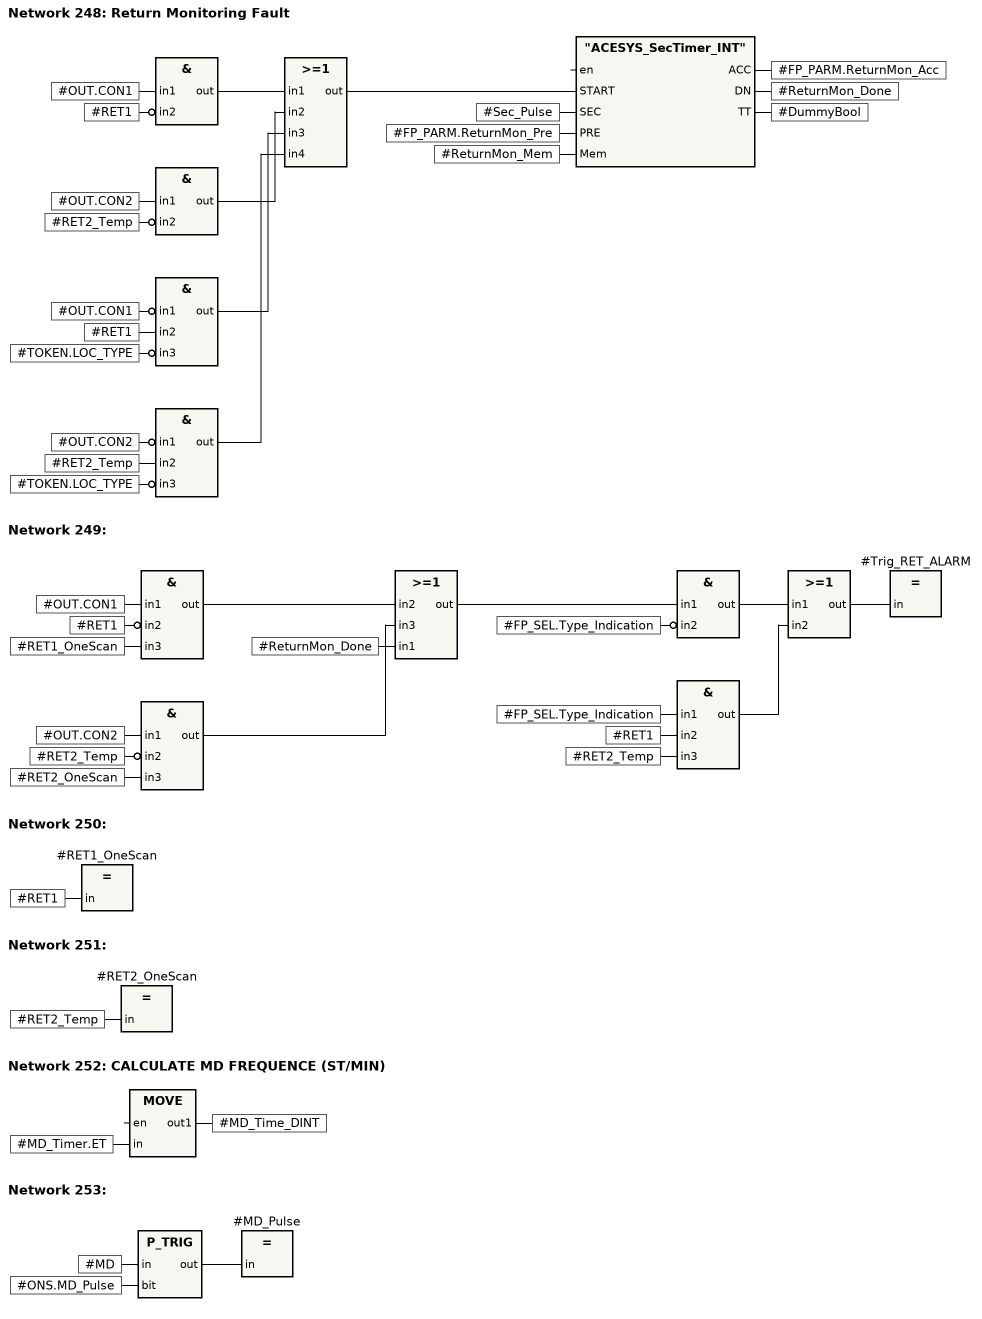
   "ACESYS_SecTimer_INT"(START := (#OUT.CON1 AND NOT #RET1) OR (#OUT.CON2 AND NOT #RET2_Temp) OR (NOT #OUT.CON1 AND #RET1 AND NOT #TOKEN.LOC_TYPE) OR (NOT #OUT.CON2 AND #RET2_Temp AND NOT #TOKEN.LOC_TYPE),
                         SEC := #Sec_Pulse,
                         PRE := #FP_PARM.ReturnMon_Pre,
                         Mem := #ReturnMon_Mem,
                         ACC => #FP_PARM.ReturnMon_Acc,
                         DN => #ReturnMon_Done,
                         TT => #DummyBool);
END_REGION

REGION Network 249
   #Trig_RET_ALARM := (((#OUT.CON1 AND NOT #RET1 AND #RET1_OneScan) OR (#OUT.CON2 AND NOT #RET2_Temp AND #RET2_OneScan) OR #ReturnMon_Done) AND NOT #FP_SEL.Type_Indication) OR (#FP_SEL.Type_Indication AND #RET1 AND #RET2_Temp);
END_REGION

REGION Network 250
   #RET1_OneScan := #RET1;
END_REGION

REGION Network 251
   #RET2_OneScan := #RET2_Temp;
END_REGION

REGION Network 252: CALCULATE MD FREQUENCE (ST/MIN)
   #MD_Time_DINT := #MD_Timer.ET;
END_REGION

REGION Network 253
   #_w1 := #MD AND NOT #ONS.MD_Pulse;   // rising edge
   #ONS.MD_Pulse := #MD;
   #MD_Pulse := #_w1;
END_REGION

REGION Network 254
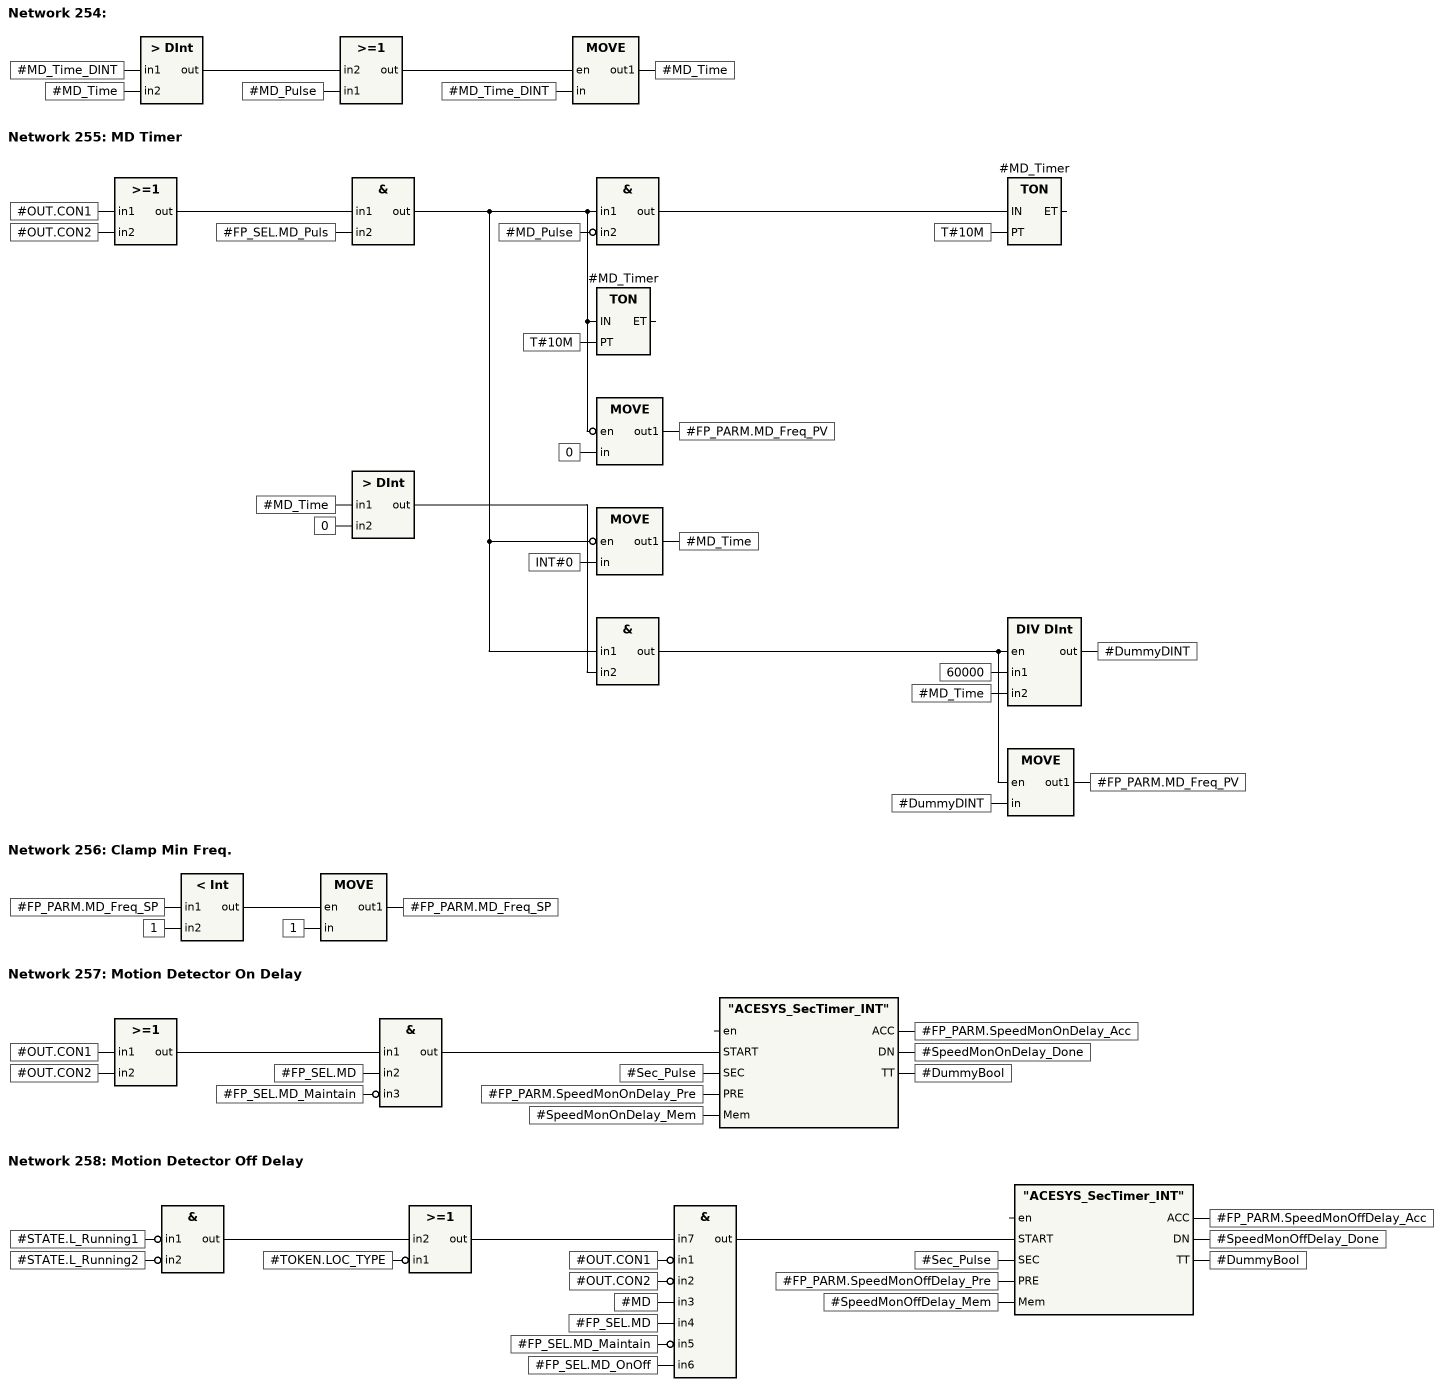
   IF (#MD_Time_DINT > #MD_Time) OR #MD_Pulse THEN #MD_Time := #MD_Time_DINT; END_IF;
END_REGION

REGION Network 255: MD Timer
   // The MD_Timer is inserted twice to ensure that the timer is enabled in the same 
   // scan after af MD pulse.
   #_w1 := (#OUT.CON1 OR #OUT.CON2) AND #FP_SEL.MD_Puls;
   #MD_Timer(IN := #_w1 AND NOT #MD_Pulse, PT := T#10M);   // TON
   #MD_Timer(IN := #_w1, PT := T#10M);   // TON
   IF NOT #_w1 THEN
       #FP_PARM.MD_Freq_PV := 0;
       #MD_Time := INT#0;
   END_IF;
   IF #_w1 AND (#MD_Time > 0) THEN
       #DummyDINT := 60000 / #MD_Time;
       #FP_PARM.MD_Freq_PV := #DummyDINT;
   END_IF;
END_REGION

REGION Network 256: Clamp Min Freq.
   IF #FP_PARM.MD_Freq_SP < 1 THEN #FP_PARM.MD_Freq_SP := 1; END_IF;
END_REGION

REGION Network 257: Motion Detector On Delay
   "ACESYS_SecTimer_INT"(START := (#OUT.CON1 OR #OUT.CON2) AND #FP_SEL.MD AND NOT #FP_SEL.MD_Maintain,
                         SEC := #Sec_Pulse,
                         PRE := #FP_PARM.SpeedMonOnDelay_Pre,
                         Mem := #SpeedMonOnDelay_Mem,
                         ACC => #FP_PARM.SpeedMonOnDelay_Acc,
                         DN => #SpeedMonOnDelay_Done,
                         TT => #DummyBool);
END_REGION

REGION Network 258: Motion Detector Off Delay
   // Build 003 - 1.July.2019 (EXTBOB): Added logic to inhibit motion fault when running in "electrical" local mode.
   "ACESYS_SecTimer_INT"(START := ((NOT #STATE.L_Running1 AND NOT #STATE.L_Running2) OR NOT #TOKEN.LOC_TYPE) AND NOT #OUT.CON1 AND NOT #OUT.CON2 AND #MD AND #FP_SEL.MD AND NOT #FP_SEL.MD_Maintain AND #FP_SEL.MD_OnOff,
                         SEC := #Sec_Pulse,
                         PRE := #FP_PARM.SpeedMonOffDelay_Pre,
                         Mem := #SpeedMonOffDelay_Mem,
                         ACC => #FP_PARM.SpeedMonOffDelay_Acc,
                         DN => #SpeedMonOffDelay_Done,
                         TT => #DummyBool);
END_REGION

REGION Network 259: Motion Detector Trig Delay
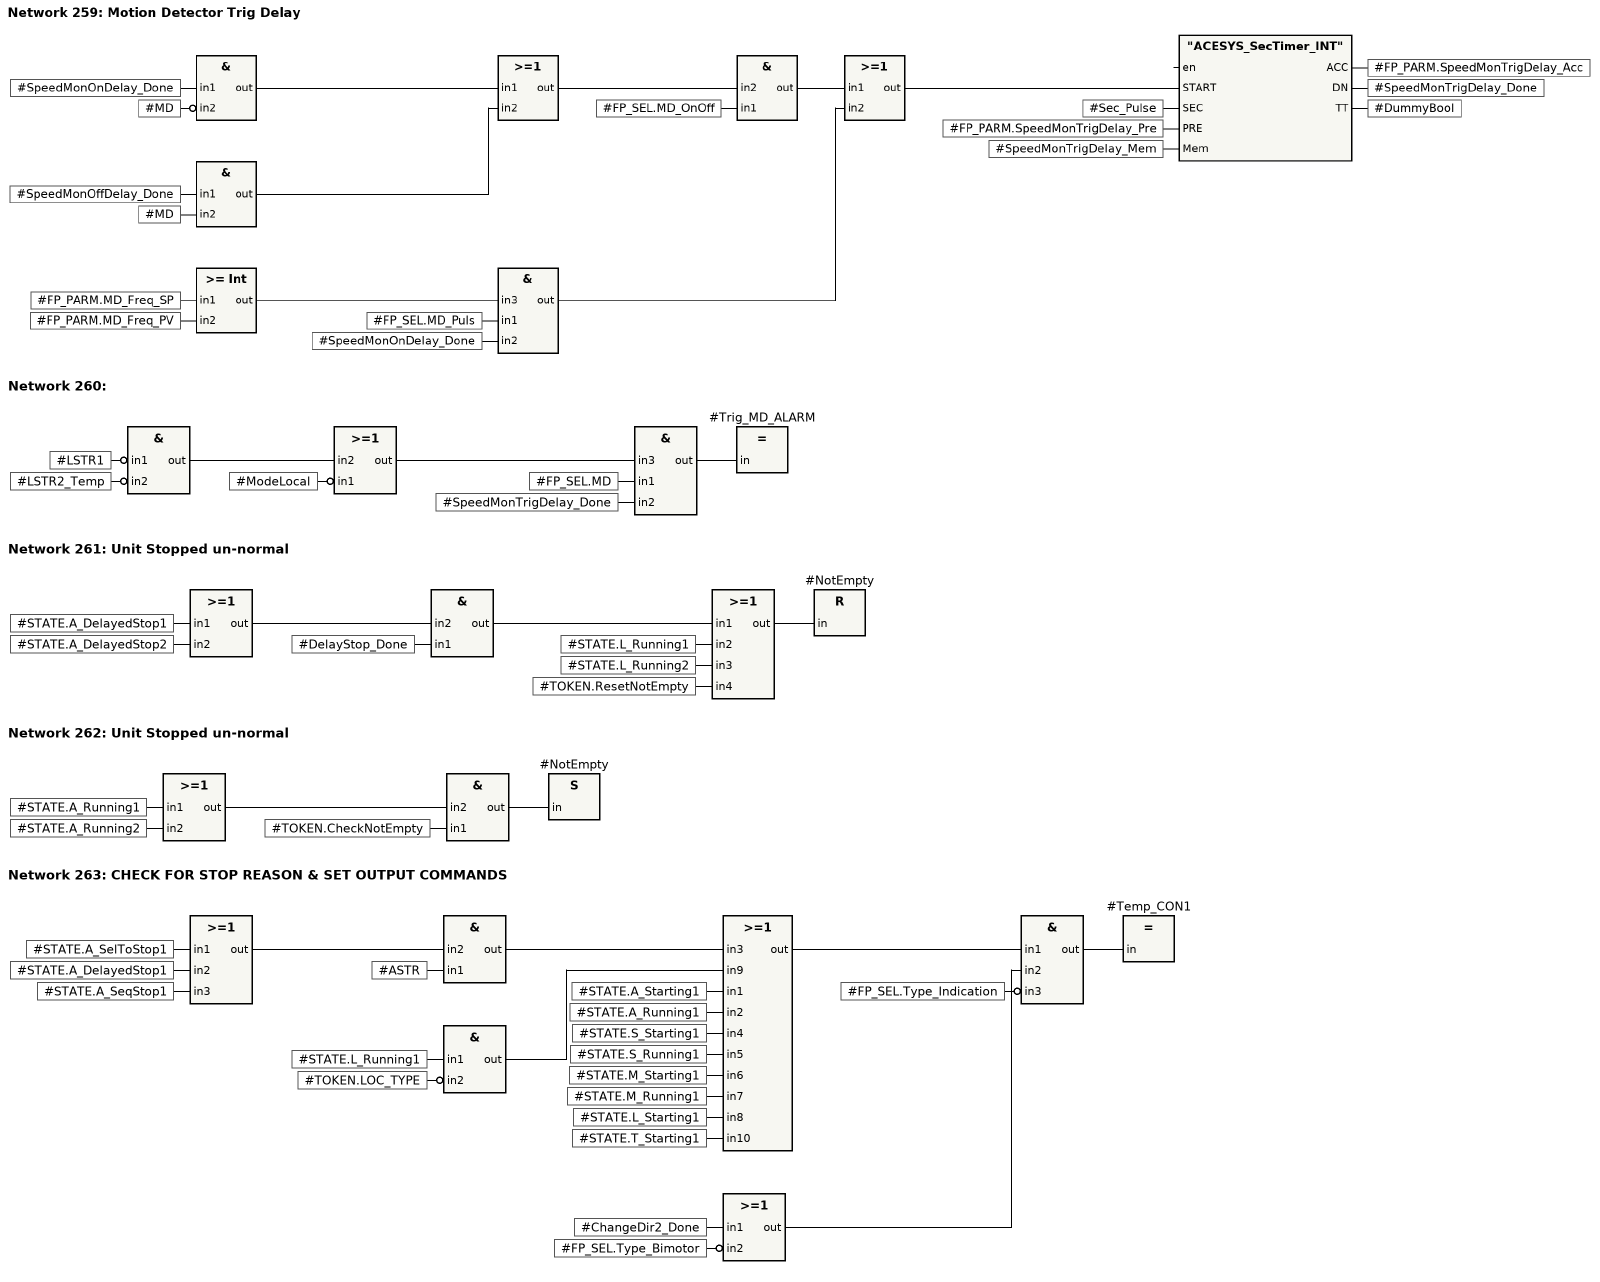
   "ACESYS_SecTimer_INT"(START := (((#SpeedMonOnDelay_Done AND NOT #MD) OR (#SpeedMonOffDelay_Done AND #MD)) AND #FP_SEL.MD_OnOff) OR ((#FP_PARM.MD_Freq_SP >= #FP_PARM.MD_Freq_PV) AND #FP_SEL.MD_Puls AND #SpeedMonOnDelay_Done),
                         SEC := #Sec_Pulse,
                         PRE := #FP_PARM.SpeedMonTrigDelay_Pre,
                         Mem := #SpeedMonTrigDelay_Mem,
                         ACC => #FP_PARM.SpeedMonTrigDelay_Acc,
                         DN => #SpeedMonTrigDelay_Done,
                         TT => #DummyBool);
END_REGION

REGION Network 260
   #Trig_MD_ALARM := ((NOT #LSTR1 AND NOT #LSTR2_Temp) OR NOT #ModeLocal) AND #FP_SEL.MD AND #SpeedMonTrigDelay_Done;
END_REGION

REGION Network 261: Unit Stopped un-normal
   // CHECK FOR MATERIANL IN LINE (NOT EMPTY)
   IF ((#STATE.A_DelayedStop1 OR #STATE.A_DelayedStop2) AND #DelayStop_Done) OR #STATE.L_Running1 OR #STATE.L_Running2 OR #TOKEN.ResetNotEmpty THEN
       #NotEmpty := FALSE;
   END_IF;
END_REGION

REGION Network 262: Unit Stopped un-normal
   // OK & INTL flags are replaced with A_Running1/2 flags
   IF (#STATE.A_Running1 OR #STATE.A_Running2) AND #TOKEN.CheckNotEmpty THEN #NotEmpty := TRUE; END_IF;
END_REGION

REGION Network 263: CHECK FOR STOP REASON & SET OUTPUT COMMANDS
   #Temp_CON1 := (((#STATE.A_SelToStop1 OR #STATE.A_DelayedStop1 OR #STATE.A_SeqStop1) AND #ASTR) OR (#STATE.L_Running1 AND NOT #TOKEN.LOC_TYPE) OR #STATE.A_Starting1 OR #STATE.A_Running1 OR #STATE.S_Starting1 OR #STATE.S_Running1 OR #STATE.M_Starting1 OR #STATE.M_Running1 OR #STATE.L_Starting1 OR #STATE.T_Starting1) AND (#ChangeDir2_Done OR NOT #FP_SEL.Type_Bimotor) AND NOT #FP_SEL.Type_Indication;
END_REGION

REGION Network 264
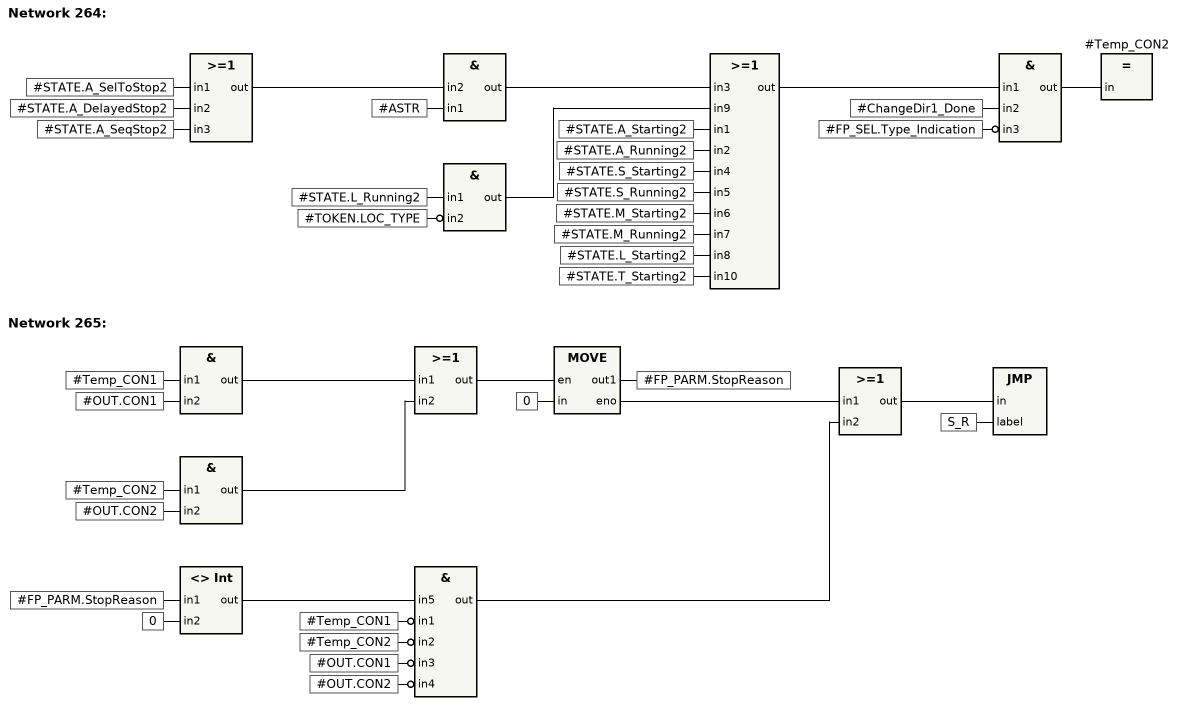
   #Temp_CON2 := (((#STATE.A_SelToStop2 OR #STATE.A_DelayedStop2 OR #STATE.A_SeqStop2) AND #ASTR) OR (#STATE.L_Running2 AND NOT #TOKEN.LOC_TYPE) OR #STATE.A_Starting2 OR #STATE.A_Running2 OR #STATE.S_Starting2 OR #STATE.S_Running2 OR #STATE.M_Starting2 OR #STATE.M_Running2 OR #STATE.L_Starting2 OR #STATE.T_Starting2) AND #ChangeDir1_Done AND NOT #FP_SEL.Type_Indication;
END_REGION

REGION Network 265
   // ENO of a box is taken as its EN; it also drops when the box reports an error
   #_w1 := (#Temp_CON1 AND #OUT.CON1) OR (#Temp_CON2 AND #OUT.CON2);
   IF #_w1 THEN #FP_PARM.StopReason := 0; END_IF;
   IF #_w1 OR ((#FP_PARM.StopReason <> 0) AND NOT #Temp_CON1 AND NOT #Temp_CON2 AND NOT #OUT.CON1 AND NOT #OUT.CON2) THEN
       GOTO S_R;
   END_IF;
END_REGION

REGION Network 266: Stop Reason
   // 0=In Operation
   // 1=Normal Stop
   // 2=Quick Stop
   // 3=Faceplate Stop
   // 4=Local Stop
   // 5=Change To Auto Mode
   // 6=Quick Stop From Unit Faceplate
   // 9=Sequence Interlock
   // 10=Interlock
   // 11=Unit Alarm
   // 12=Emergency Stop
   // 99=Unknown Reason
   // 
   // Build 003 - 8.July.2019 (EXTBOB): Stop Reason when ASTR goes low implemented
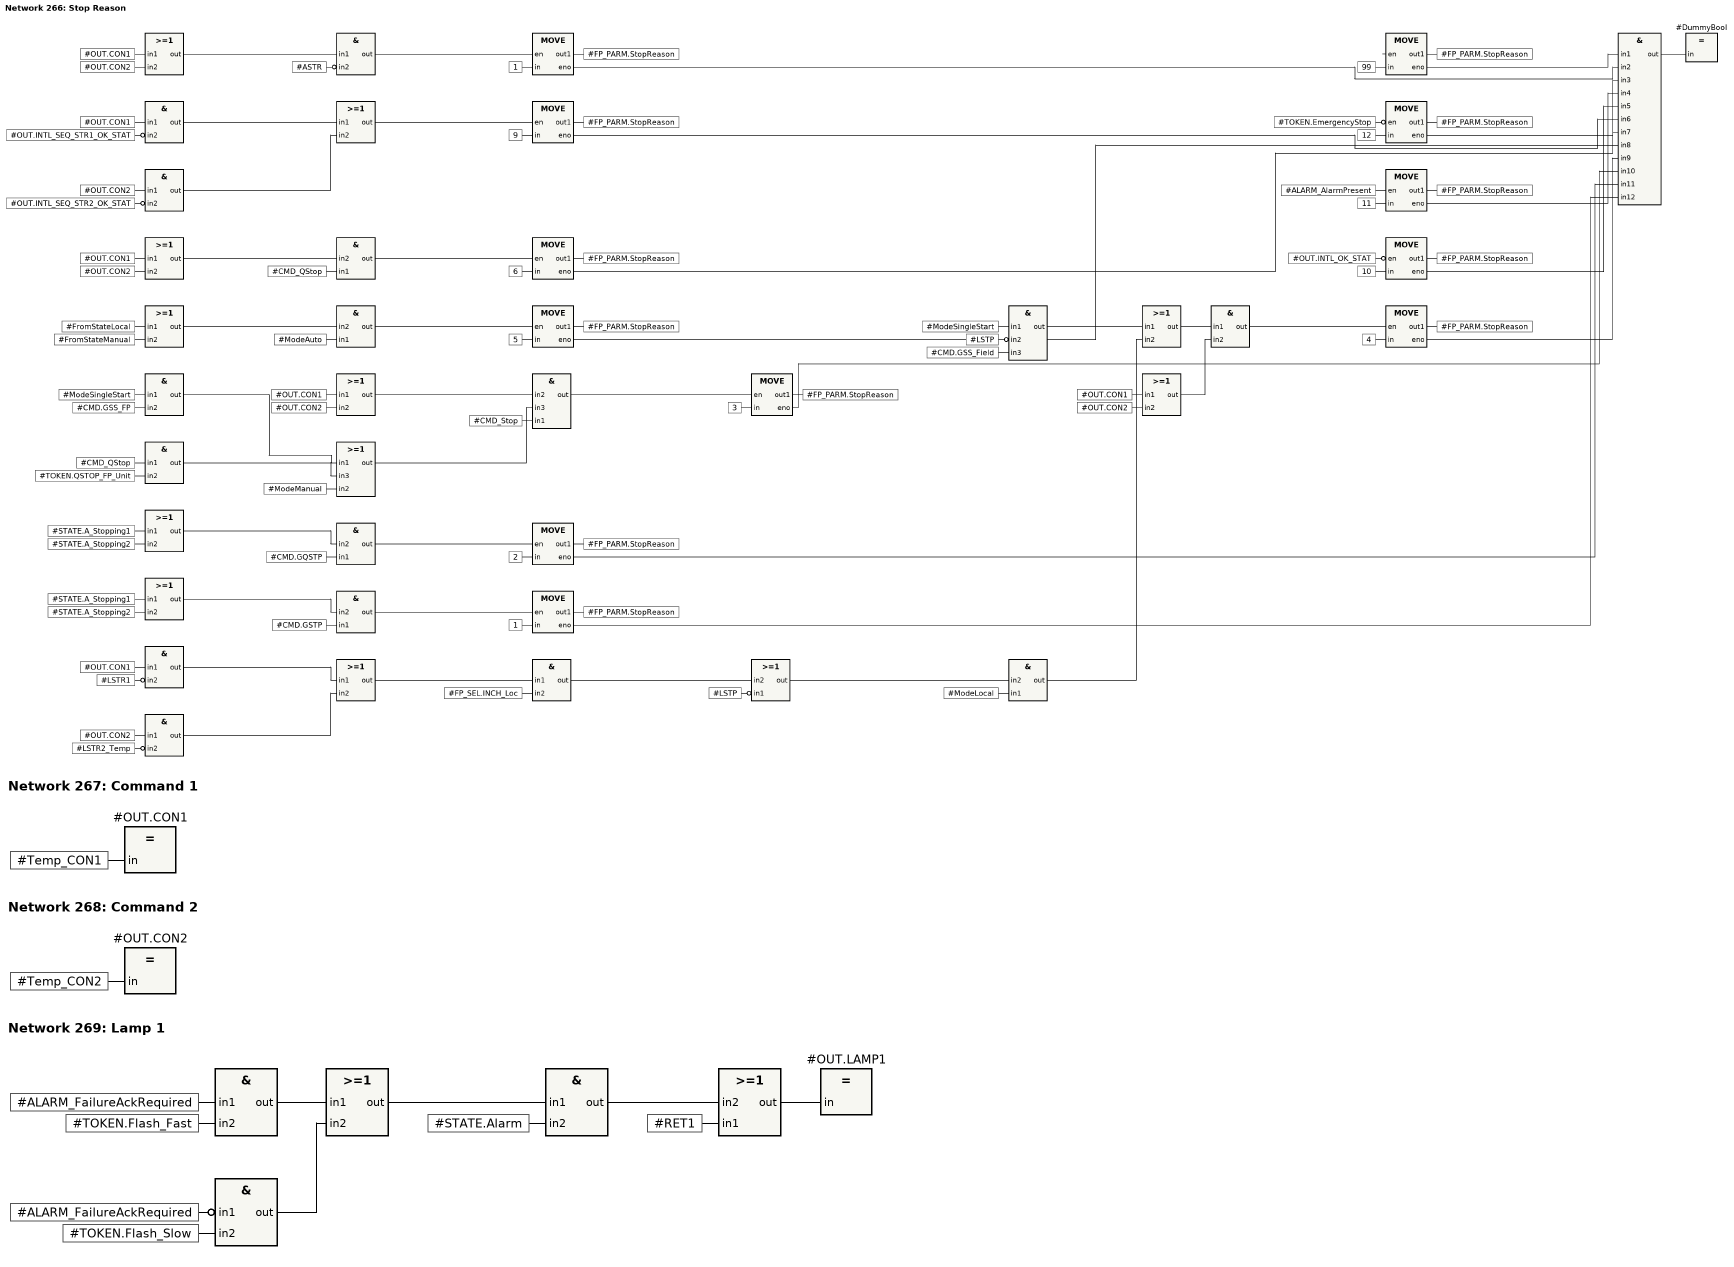
   // ENO of a box is taken as its EN; it also drops when the box reports an error
   #FP_PARM.StopReason := 99;
   #_w1 := (#OUT.CON1 OR #OUT.CON2) AND NOT #ASTR;
   IF #_w1 THEN #FP_PARM.StopReason := 1; END_IF;
   IF NOT #TOKEN.EmergencyStop THEN #FP_PARM.StopReason := 12; END_IF;
   IF #ALARM_AlarmPresent THEN #FP_PARM.StopReason := 11; END_IF;
   IF NOT #OUT.INTL_OK_STAT THEN #FP_PARM.StopReason := 10; END_IF;
   #_w2 := (#OUT.CON1 AND NOT #OUT.INTL_SEQ_STR1_OK_STAT) OR (#OUT.CON2 AND NOT #OUT.INTL_SEQ_STR2_OK_STAT);
   IF #_w2 THEN #FP_PARM.StopReason := 9; END_IF;
   #_w3 := (#OUT.CON1 OR #OUT.CON2) AND #CMD_QStop;
   IF #_w3 THEN #FP_PARM.StopReason := 6; END_IF;
   #_w4 := (#FromStateLocal OR #FromStateManual) AND #ModeAuto;
   IF #_w4 THEN #FP_PARM.StopReason := 5; END_IF;
   #_w5 := ((#ModeSingleStart AND NOT #LSTP AND #CMD.GSS_Field) OR (((((#OUT.CON1 AND NOT #LSTR1) OR (#OUT.CON2 AND NOT #LSTR2_Temp)) AND #FP_SEL.INCH_Loc) OR NOT #LSTP) AND #ModeLocal)) AND (#OUT.CON1 OR #OUT.CON2);
   IF #_w5 THEN #FP_PARM.StopReason := 4; END_IF;
   #_w6 := (#OUT.CON1 OR #OUT.CON2) AND ((#ModeSingleStart AND #CMD.GSS_FP) OR (#CMD_QStop AND #TOKEN.QSTOP_FP_Unit) OR #ModeManual) AND #CMD_Stop;
   IF #_w6 THEN #FP_PARM.StopReason := 3; END_IF;
   #_w7 := (#STATE.A_Stopping1 OR #STATE.A_Stopping2) AND #CMD.GQSTP;
   IF #_w7 THEN #FP_PARM.StopReason := 2; END_IF;
   #_w8 := (#STATE.A_Stopping1 OR #STATE.A_Stopping2) AND #CMD.GSTP;
   IF #_w8 THEN #FP_PARM.StopReason := 1; END_IF;
   #DummyBool := #_w1 AND NOT #TOKEN.EmergencyStop AND #ALARM_AlarmPresent AND NOT #OUT.INTL_OK_STAT AND #_w2 AND #_w3 AND #_w4 AND #_w5 AND #_w6 AND #_w7 AND #_w8;
END_REGION

REGION Network 267: Command 1
   S_R:
   #OUT.CON1 := #Temp_CON1;
END_REGION

REGION Network 268: Command 2
   #OUT.CON2 := #Temp_CON2;
END_REGION

REGION Network 269: Lamp 1
   // OUTPUT
   #OUT.LAMP1 := (((#ALARM_FailureAckRequired AND #TOKEN.Flash_Fast) OR (NOT #ALARM_FailureAckRequired AND #TOKEN.Flash_Slow)) AND #STATE.Alarm) OR #RET1;
END_REGION

REGION Network 270: Lamp 2
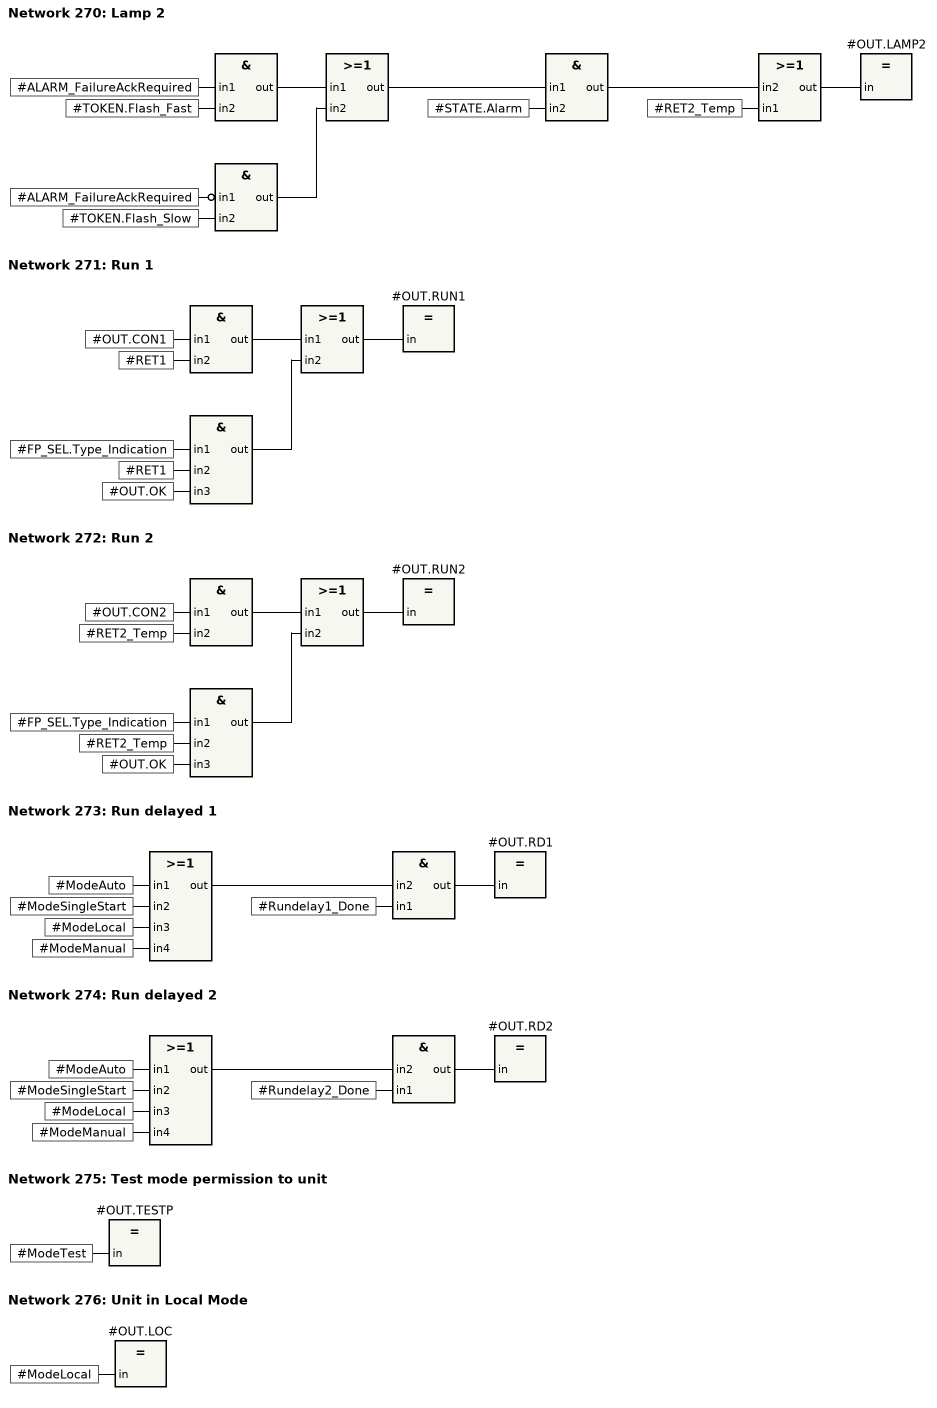
   #OUT.LAMP2 := (((#ALARM_FailureAckRequired AND #TOKEN.Flash_Fast) OR (NOT #ALARM_FailureAckRequired AND #TOKEN.Flash_Slow)) AND #STATE.Alarm) OR #RET2_Temp;
END_REGION

REGION Network 271: Run 1
   #OUT.RUN1 := (#OUT.CON1 AND #RET1) OR (#FP_SEL.Type_Indication AND #RET1 AND #OUT.OK);
END_REGION

REGION Network 272: Run 2
   #OUT.RUN2 := (#OUT.CON2 AND #RET2_Temp) OR (#FP_SEL.Type_Indication AND #RET2_Temp AND #OUT.OK);
END_REGION

REGION Network 273: Run delayed 1
   #OUT.RD1 := (#ModeAuto OR #ModeSingleStart OR #ModeLocal OR #ModeManual) AND #Rundelay1_Done;
END_REGION

REGION Network 274: Run delayed 2
   #OUT.RD2 := (#ModeAuto OR #ModeSingleStart OR #ModeLocal OR #ModeManual) AND #Rundelay2_Done;
END_REGION

REGION Network 275: Test mode permission to unit
   #OUT.TESTP := #ModeTest;
END_REGION

REGION Network 276: Unit in Local Mode
   #OUT.LOC := #ModeLocal;
END_REGION

REGION Network 277: Unit in Manual Mode
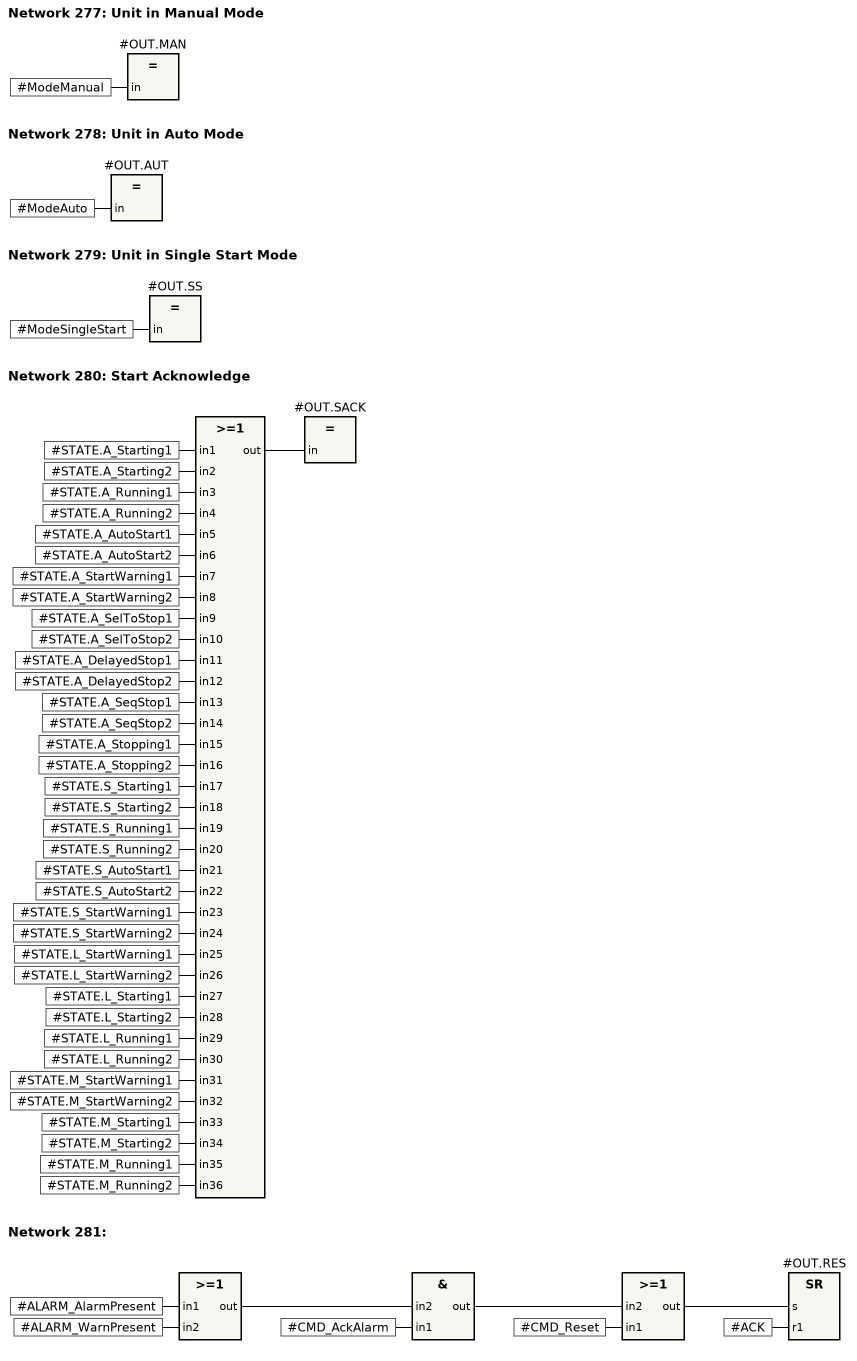
   #OUT.MAN := #ModeManual;
END_REGION

REGION Network 278: Unit in Auto Mode
   #OUT.AUT := #ModeAuto;
END_REGION

REGION Network 279: Unit in Single Start Mode
   #OUT.SS := #ModeSingleStart;
END_REGION

REGION Network 280: Start Acknowledge
   #OUT.SACK := #STATE.A_Starting1 OR #STATE.A_Starting2 OR #STATE.A_Running1 OR #STATE.A_Running2 OR #STATE.A_AutoStart1 OR #STATE.A_AutoStart2 OR #STATE.A_StartWarning1 OR #STATE.A_StartWarning2 OR #STATE.A_SelToStop1 OR #STATE.A_SelToStop2 OR #STATE.A_DelayedStop1 OR #STATE.A_DelayedStop2 OR #STATE.A_SeqStop1 OR #STATE.A_SeqStop2 OR #STATE.A_Stopping1 OR #STATE.A_Stopping2 OR #STATE.S_Starting1 OR #STATE.S_Starting2 OR #STATE.S_Running1 OR #STATE.S_Running2 OR #STATE.S_AutoStart1 OR #STATE.S_AutoStart2 OR #STATE.S_StartWarning1 OR #STATE.S_StartWarning2 OR #STATE.L_StartWarning1 OR #STATE.L_StartWarning2 OR #STATE.L_Starting1 OR #STATE.L_Starting2 OR #STATE.L_Running1 OR #STATE.L_Running2 OR #STATE.M_StartWarning1 OR #STATE.M_StartWarning2 OR #STATE.M_Starting1 OR #STATE.M_Starting2 OR #STATE.M_Running1 OR #STATE.M_Running2;
END_REGION

REGION Network 281
   IF ((#ALARM_AlarmPresent OR #ALARM_WarnPresent) AND #CMD_AckAlarm) OR #CMD_Reset THEN
       #OUT.RES := TRUE;   // SR flip-flop
   END_IF;
   IF #ACK THEN #OUT.RES := FALSE; END_IF;
END_REGION

REGION Network 282: Unit Status OK (no alarms)
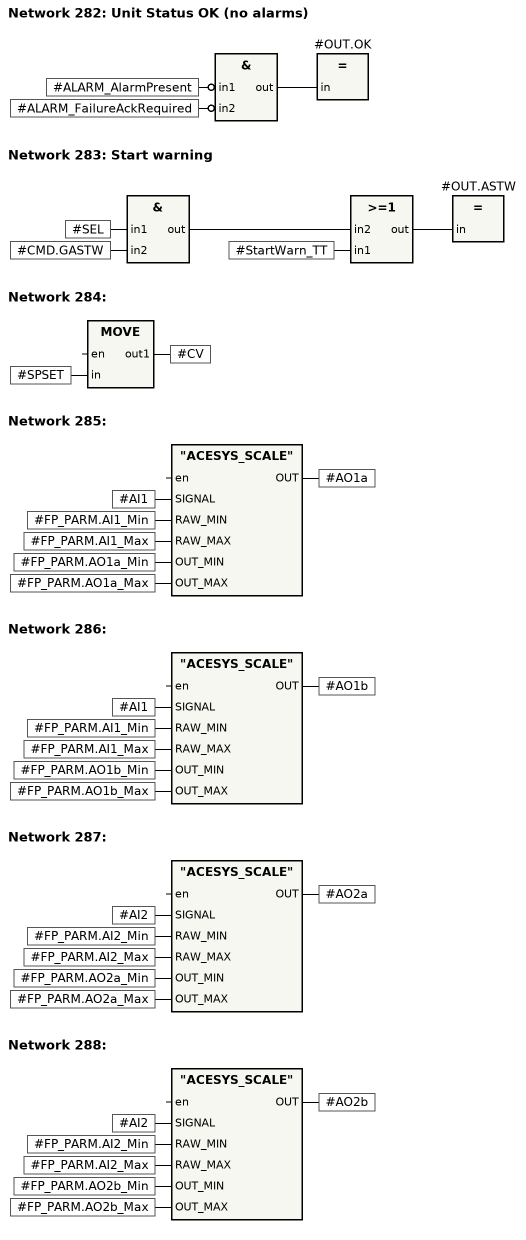
   #OUT.OK := NOT #ALARM_AlarmPresent AND NOT #ALARM_FailureAckRequired;
END_REGION

REGION Network 283: Start warning
   #OUT.ASTW := (#SEL AND #CMD.GASTW) OR #StartWarn_TT;
END_REGION

REGION Network 284
   #CV := #SPSET;
END_REGION

REGION Network 285
   "ACESYS_SCALE"(SIGNAL := #AI1,
                  RAW_MIN := #FP_PARM.AI1_Min,
                  RAW_MAX := #FP_PARM.AI1_Max,
                  OUT_MIN := #FP_PARM.AO1a_Min,
                  OUT_MAX := #FP_PARM.AO1a_Max,
                  OUT => #AO1a);
END_REGION

REGION Network 286
   "ACESYS_SCALE"(SIGNAL := #AI1,
                  RAW_MIN := #FP_PARM.AI1_Min,
                  RAW_MAX := #FP_PARM.AI1_Max,
                  OUT_MIN := #FP_PARM.AO1b_Min,
                  OUT_MAX := #FP_PARM.AO1b_Max,
                  OUT => #AO1b);
END_REGION

REGION Network 287
   "ACESYS_SCALE"(SIGNAL := #AI2,
                  RAW_MIN := #FP_PARM.AI2_Min,
                  RAW_MAX := #FP_PARM.AI2_Max,
                  OUT_MIN := #FP_PARM.AO2a_Min,
                  OUT_MAX := #FP_PARM.AO2a_Max,
                  OUT => #AO2a);
END_REGION

REGION Network 288
   "ACESYS_SCALE"(SIGNAL := #AI2,
                  RAW_MIN := #FP_PARM.AI2_Min,
                  RAW_MAX := #FP_PARM.AI2_Max,
                  OUT_MIN := #FP_PARM.AO2b_Min,
                  OUT_MAX := #FP_PARM.AO2b_Max,
                  OUT => #AO2b);
END_REGION

REGION Network 289
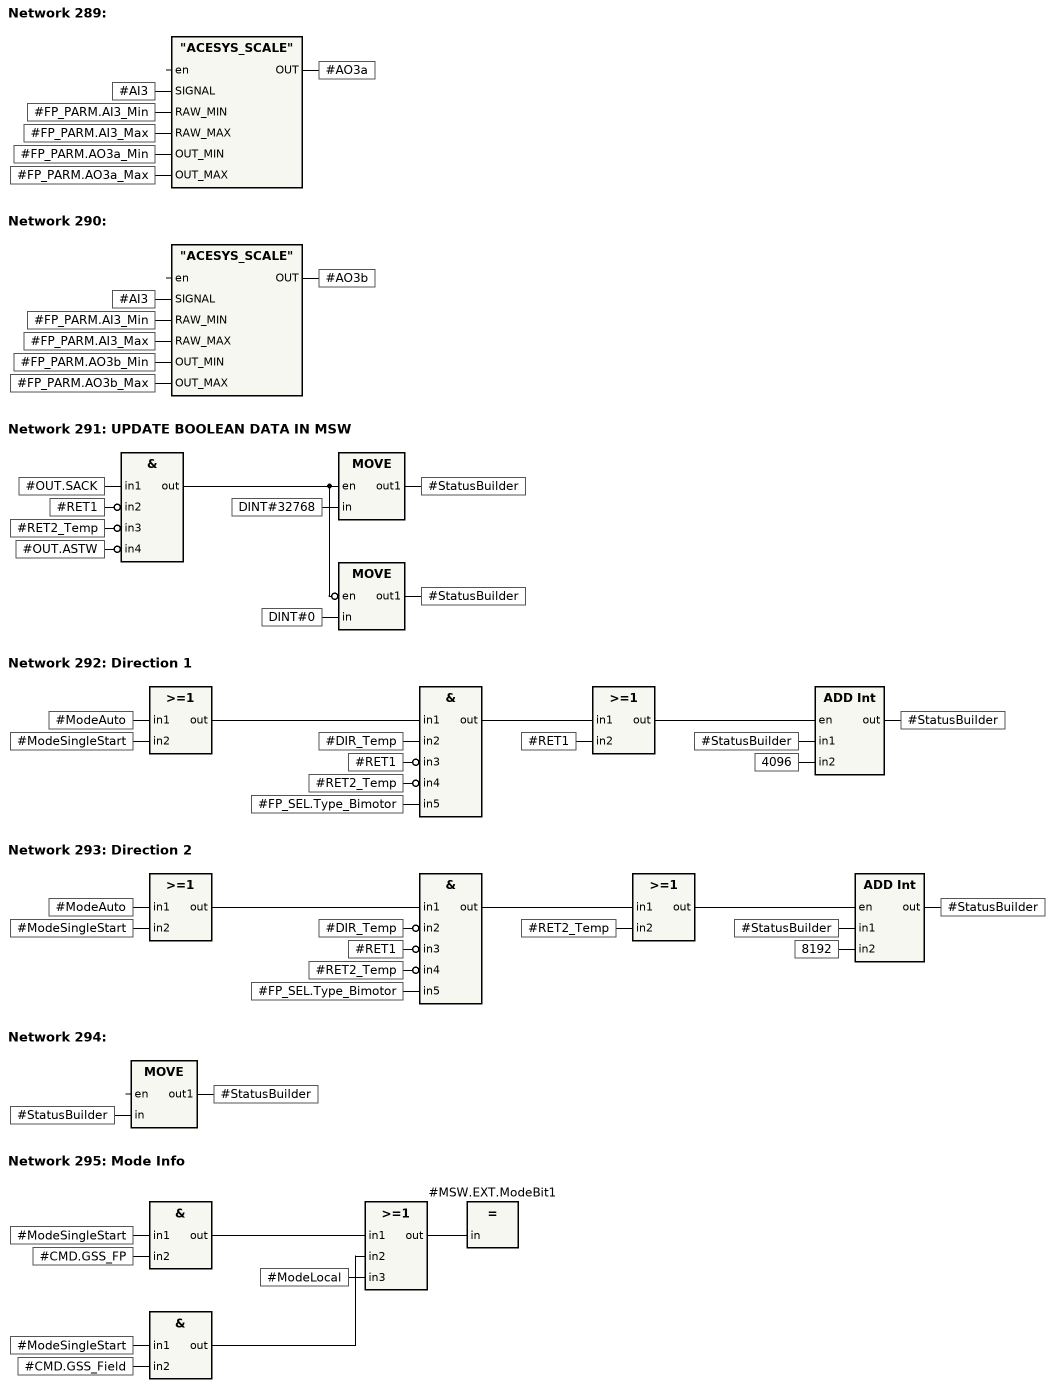
   "ACESYS_SCALE"(SIGNAL := #AI3,
                  RAW_MIN := #FP_PARM.AI3_Min,
                  RAW_MAX := #FP_PARM.AI3_Max,
                  OUT_MIN := #FP_PARM.AO3a_Min,
                  OUT_MAX := #FP_PARM.AO3a_Max,
                  OUT => #AO3a);
END_REGION

REGION Network 290
   "ACESYS_SCALE"(SIGNAL := #AI3,
                  RAW_MIN := #FP_PARM.AI3_Min,
                  RAW_MAX := #FP_PARM.AI3_Max,
                  OUT_MIN := #FP_PARM.AO3b_Min,
                  OUT_MAX := #FP_PARM.AO3b_Max,
                  OUT => #AO3b);
END_REGION

REGION Network 291: UPDATE BOOLEAN DATA IN MSW
   #_w1 := #OUT.SACK AND NOT #RET1 AND NOT #RET2_Temp AND NOT #OUT.ASTW;
   IF #_w1 THEN #StatusBuilder := DINT#32768; END_IF;
   IF NOT #_w1 THEN #StatusBuilder := DINT#0; END_IF;
END_REGION

REGION Network 292: Direction 1
   // Build 002 - 27 March 2019 - FP_Sel.Type_Bimotor Added
   IF ((#ModeAuto OR #ModeSingleStart) AND #DIR_Temp AND NOT #RET1 AND NOT #RET2_Temp AND #FP_SEL.Type_Bimotor) OR #RET1 THEN
       #StatusBuilder := #StatusBuilder + 4096;
   END_IF;
END_REGION

REGION Network 293: Direction 2
   // Build 002 - 27 March 2019 - FP_Sel.Type_Bimotor Added
   IF ((#ModeAuto OR #ModeSingleStart) AND NOT #DIR_Temp AND NOT #RET1 AND NOT #RET2_Temp AND #FP_SEL.Type_Bimotor) OR #RET2_Temp THEN
       #StatusBuilder := #StatusBuilder + 8192;
   END_IF;
END_REGION

REGION Network 294
   #StatusBuilder := #StatusBuilder;
END_REGION

REGION Network 295: Mode Info
   #MSW.EXT.ModeBit1 := (#ModeSingleStart AND #CMD.GSS_FP) OR (#ModeSingleStart AND #CMD.GSS_Field) OR #ModeLocal;
END_REGION

REGION Network 296: Mode Info
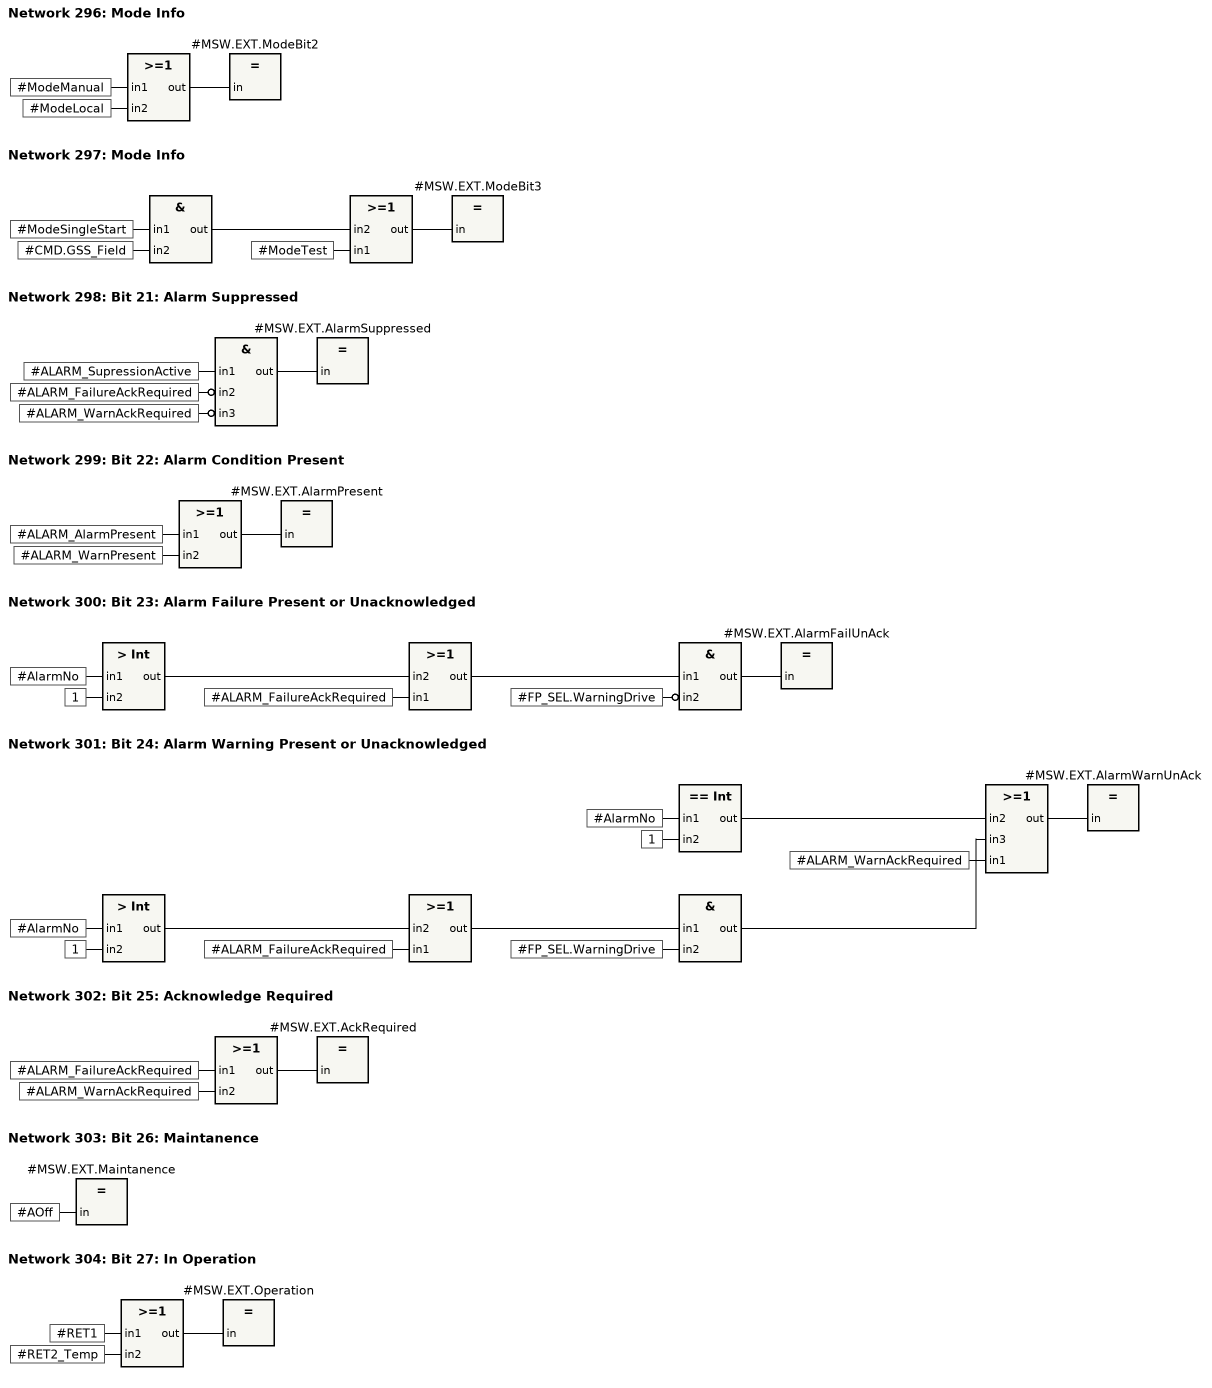
   #MSW.EXT.ModeBit2 := #ModeManual OR #ModeLocal;
END_REGION

REGION Network 297: Mode Info
   #MSW.EXT.ModeBit3 := (#ModeSingleStart AND #CMD.GSS_Field) OR #ModeTest;
END_REGION

REGION Network 298: Bit 21: Alarm Suppressed
   #MSW.EXT.AlarmSuppressed := #ALARM_SupressionActive AND NOT #ALARM_FailureAckRequired AND NOT #ALARM_WarnAckRequired;
END_REGION

REGION Network 299: Bit 22: Alarm Condition Present
   #MSW.EXT.AlarmPresent := #ALARM_AlarmPresent OR #ALARM_WarnPresent;
END_REGION

REGION Network 300: Bit 23: Alarm Failure Present or Unacknowledged
   #MSW.EXT.AlarmFailUnAck := ((#AlarmNo > 1) OR #ALARM_FailureAckRequired) AND NOT #FP_SEL.WarningDrive;
END_REGION

REGION Network 301: Bit 24: Alarm Warning Present or Unacknowledged
   #MSW.EXT.AlarmWarnUnAck := (#AlarmNo = 1) OR (((#AlarmNo > 1) OR #ALARM_FailureAckRequired) AND #FP_SEL.WarningDrive) OR #ALARM_WarnAckRequired;
END_REGION

REGION Network 302: Bit 25: Acknowledge Required
   #MSW.EXT.AckRequired := #ALARM_FailureAckRequired OR #ALARM_WarnAckRequired;
END_REGION

REGION Network 303: Bit 26: Maintanence
   #MSW.EXT.Maintanence := #AOff;
END_REGION

REGION Network 304: Bit 27: In Operation
   #MSW.EXT.Operation := #RET1 OR #RET2_Temp;
END_REGION

REGION Network 305: Bit 28: Forced
   // Build 002 - 25 March 2019 : Out of Service flag would set the Forced flag to 
   // symbols
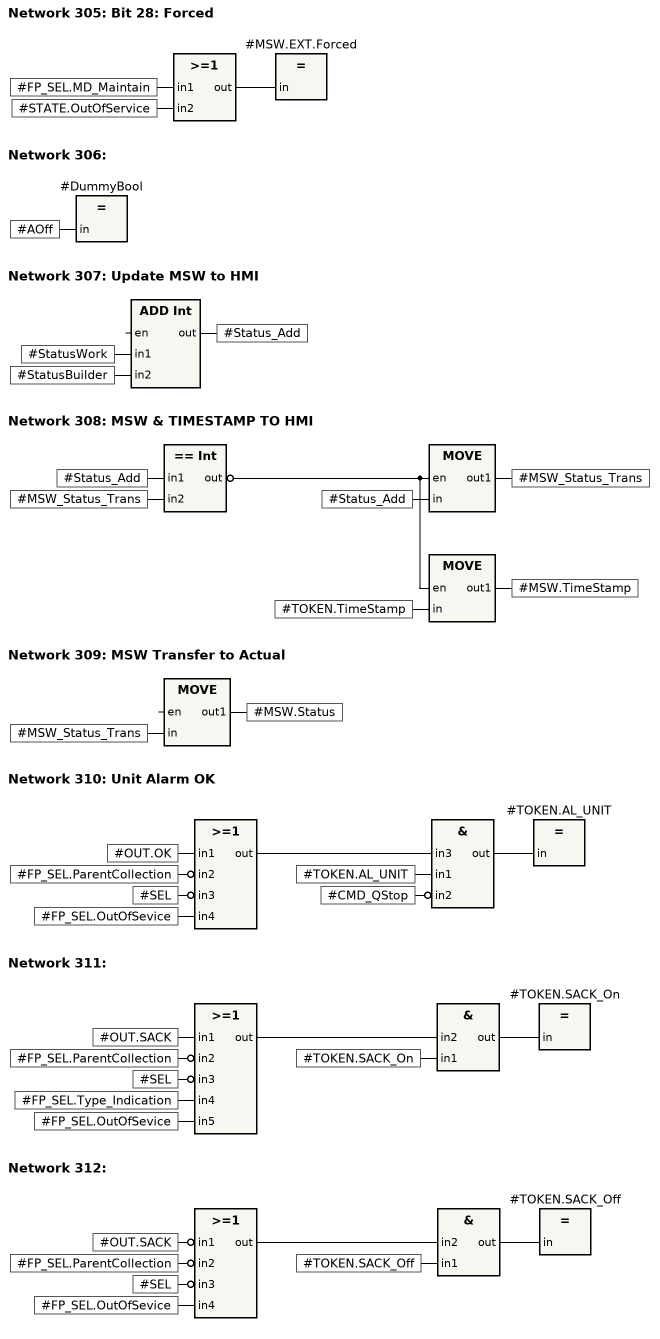
   #MSW.EXT.Forced := #FP_SEL.MD_Maintain OR #STATE.OutOfService;
END_REGION

REGION Network 306
   Done:
   #DummyBool := #AOff;
END_REGION

REGION Network 307: Update MSW to HMI
   #Status_Add := #StatusWork + #StatusBuilder;
END_REGION

REGION Network 308: MSW & TIMESTAMP TO HMI
   #_w1 := NOT (#Status_Add = #MSW_Status_Trans);
   IF #_w1 THEN
       #MSW_Status_Trans := #Status_Add;
       #MSW.TimeStamp := #TOKEN.TimeStamp;
   END_IF;
END_REGION

REGION Network 309: MSW Transfer to Actual
   #MSW.Status := #MSW_Status_Trans;
END_REGION

REGION Network 310: Unit Alarm OK
   #TOKEN.AL_UNIT := (#OUT.OK OR NOT #FP_SEL.ParentCollection OR NOT #SEL OR #FP_SEL.OutOfSevice) AND #TOKEN.AL_UNIT AND NOT #CMD_QStop;
END_REGION

REGION Network 311
   // Build 003 - 1.July.2019 (EXTBOB): Replaced "Select" with original explicit definition
   // Build 009 - 24.Jun.2020 (MIA-US): Remove CMD.GSEL
   #TOKEN.SACK_On := (#OUT.SACK OR NOT #FP_SEL.ParentCollection OR NOT #SEL OR #FP_SEL.Type_Indication OR #FP_SEL.OutOfSevice) AND #TOKEN.SACK_On;
END_REGION

REGION Network 312
   #TOKEN.SACK_Off := (NOT #OUT.SACK OR NOT #FP_SEL.ParentCollection OR NOT #SEL OR #FP_SEL.OutOfSevice) AND #TOKEN.SACK_Off;
END_REGION

REGION Network 313
   // Build 003 - 1.July.2019 (EXTBOB): Replaced "Select" with original explicit definition
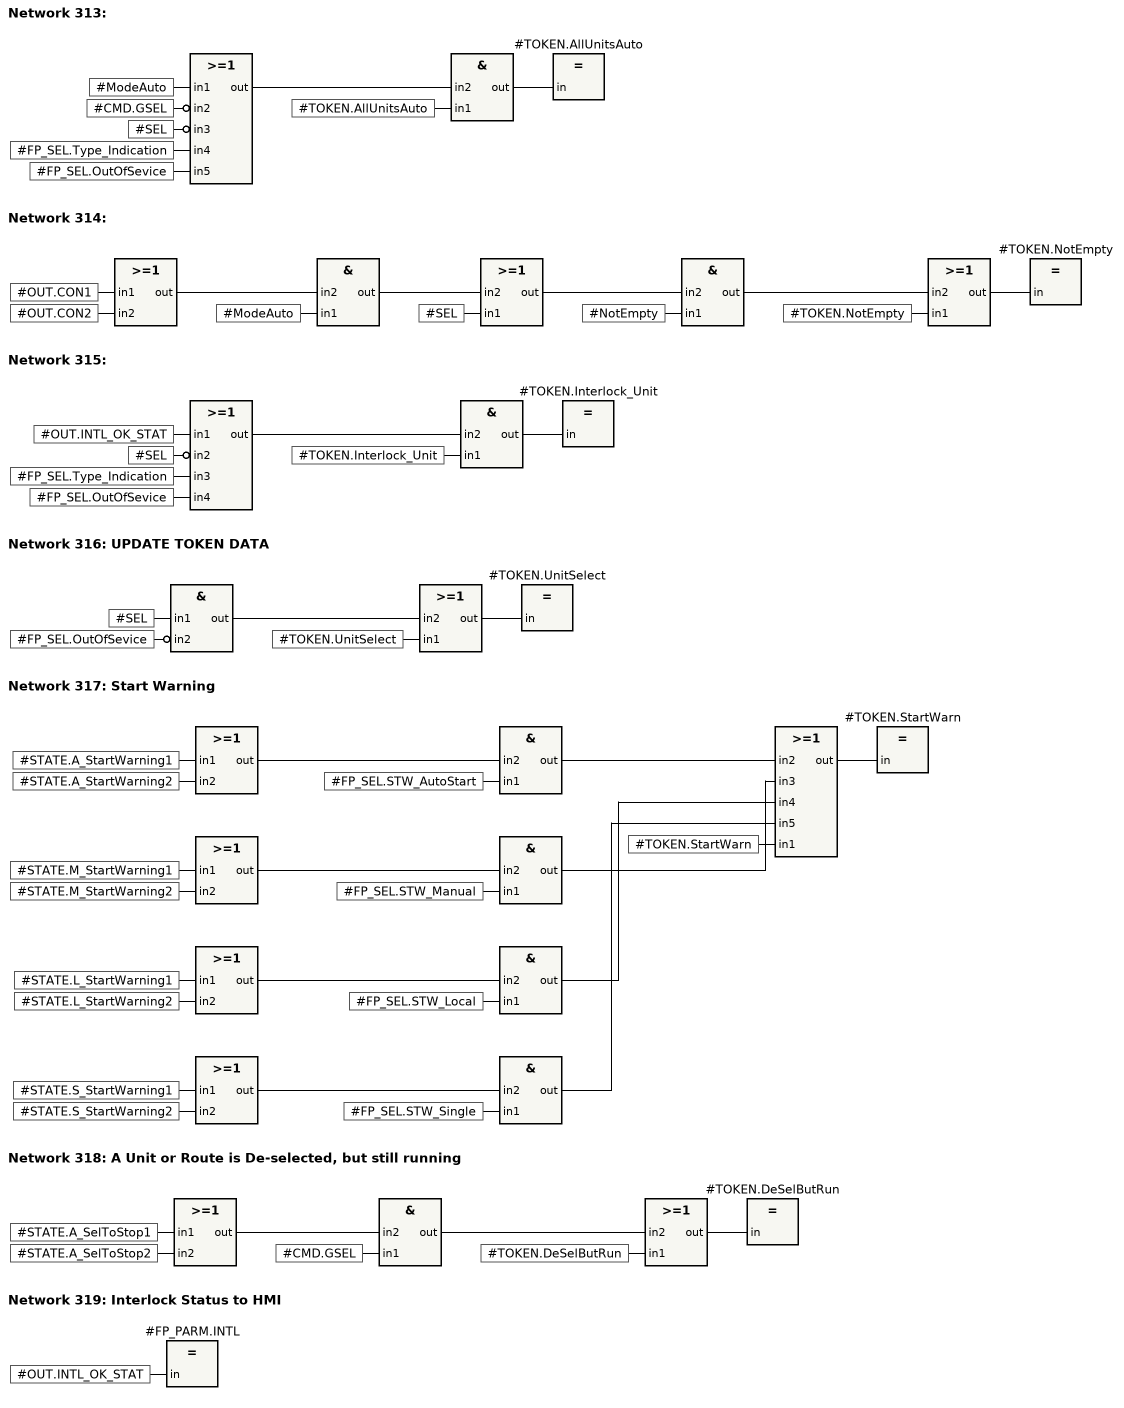
   #TOKEN.AllUnitsAuto := (#ModeAuto OR NOT #CMD.GSEL OR NOT #SEL OR #FP_SEL.Type_Indication OR #FP_SEL.OutOfSevice) AND #TOKEN.AllUnitsAuto;
END_REGION

REGION Network 314
   #TOKEN.NotEmpty := ((((#OUT.CON1 OR #OUT.CON2) AND #ModeAuto) OR #SEL) AND #NotEmpty) OR #TOKEN.NotEmpty;
END_REGION

REGION Network 315
   // Build 003 - 1.July.2019 (EXTBOB): Replaced "Select" with original explicit definition
   // Build 011 - 09.10.2020 (EXTBOB): Removed CMD.GSEL neg in OR logic to pass Intl status also in grp deselected cond in auto mode
   #TOKEN.Interlock_Unit := (#OUT.INTL_OK_STAT OR NOT #SEL OR #FP_SEL.Type_Indication OR #FP_SEL.OutOfSevice) AND #TOKEN.Interlock_Unit;
END_REGION

REGION Network 316: UPDATE TOKEN DATA
   #TOKEN.UnitSelect := (#SEL AND NOT #FP_SEL.OutOfSevice) OR #TOKEN.UnitSelect;
END_REGION

REGION Network 317: Start Warning
   #TOKEN.StartWarn := ((#STATE.A_StartWarning1 OR #STATE.A_StartWarning2) AND #FP_SEL.STW_AutoStart) OR ((#STATE.M_StartWarning1 OR #STATE.M_StartWarning2) AND #FP_SEL.STW_Manual) OR ((#STATE.L_StartWarning1 OR #STATE.L_StartWarning2) AND #FP_SEL.STW_Local) OR ((#STATE.S_StartWarning1 OR #STATE.S_StartWarning2) AND #FP_SEL.STW_Single) OR #TOKEN.StartWarn;
END_REGION

REGION Network 318: A Unit or Route is De-selected, but still running
   #TOKEN.DeSelButRun := ((#STATE.A_SelToStop1 OR #STATE.A_SelToStop2) AND #CMD.GSEL) OR #TOKEN.DeSelButRun;
END_REGION

REGION Network 319: Interlock Status to HMI
   #FP_PARM.INTL := #OUT.INTL_OK_STAT;
END_REGION

REGION Network 320: Interlock Status to HMI
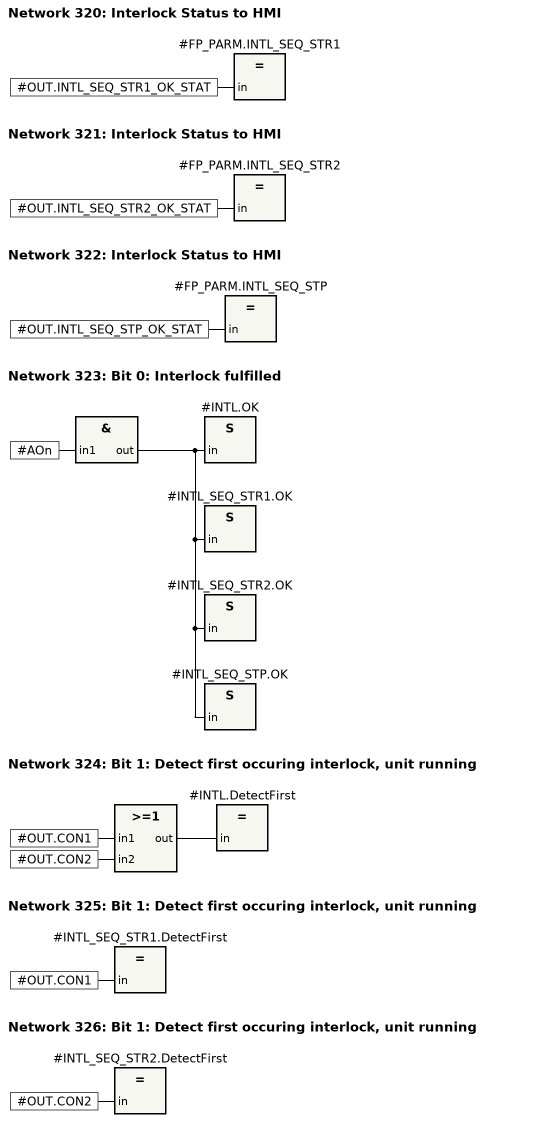
   #FP_PARM.INTL_SEQ_STR1 := #OUT.INTL_SEQ_STR1_OK_STAT;
END_REGION

REGION Network 321: Interlock Status to HMI
   #FP_PARM.INTL_SEQ_STR2 := #OUT.INTL_SEQ_STR2_OK_STAT;
END_REGION

REGION Network 322: Interlock Status to HMI
   #FP_PARM.INTL_SEQ_STP := #OUT.INTL_SEQ_STP_OK_STAT;
END_REGION

REGION Network 323: Bit 0: Interlock fulfilled
   // INTERLOCK LINK
   IF #AOn THEN
       #INTL.OK := TRUE;
       #INTL_SEQ_STR1.OK := TRUE;
       #INTL_SEQ_STR2.OK := TRUE;
       #INTL_SEQ_STP.OK := TRUE;
   END_IF;
END_REGION

REGION Network 324: Bit 1: Detect first occuring interlock, unit running
   #INTL.DetectFirst := #OUT.CON1 OR #OUT.CON2;
END_REGION

REGION Network 325: Bit 1: Detect first occuring interlock, unit running
   #INTL_SEQ_STR1.DetectFirst := #OUT.CON1;
END_REGION

REGION Network 326: Bit 1: Detect first occuring interlock, unit running
   #INTL_SEQ_STR2.DetectFirst := #OUT.CON2;
END_REGION

REGION Network 327: Bit 3: Clear first Interlock
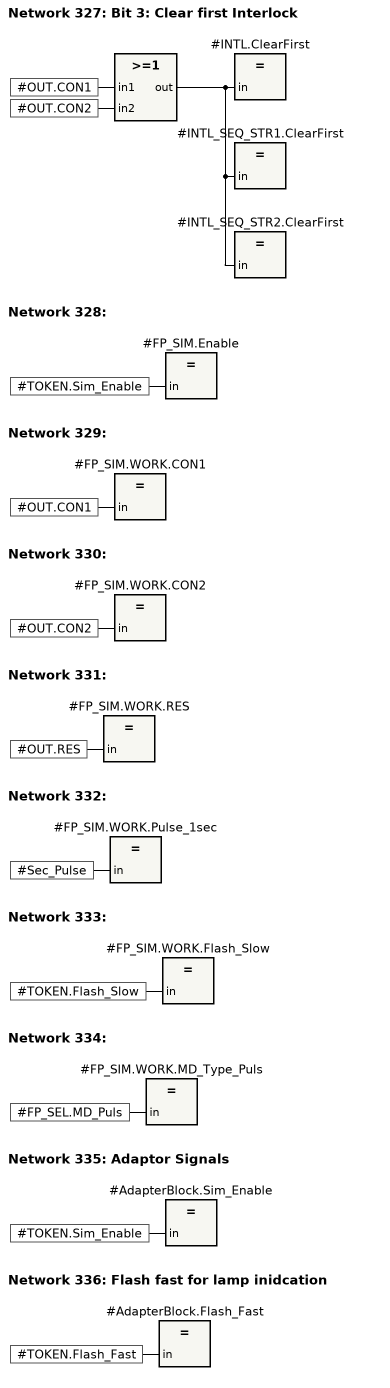
   #INTL.ClearFirst := #OUT.CON1 OR #OUT.CON2;
   #INTL_SEQ_STR1.ClearFirst := #INTL.ClearFirst;
   #INTL_SEQ_STR2.ClearFirst := #INTL.ClearFirst;
END_REGION

REGION Network 328
   #FP_SIM.Enable := #TOKEN.Sim_Enable;
END_REGION

REGION Network 329
   #FP_SIM.WORK.CON1 := #OUT.CON1;
END_REGION

REGION Network 330
   #FP_SIM.WORK.CON2 := #OUT.CON2;
END_REGION

REGION Network 331
   #FP_SIM.WORK.RES := #OUT.RES;
END_REGION

REGION Network 332
   #FP_SIM.WORK.Pulse_1sec := #Sec_Pulse;
END_REGION

REGION Network 333
   #FP_SIM.WORK.Flash_Slow := #TOKEN.Flash_Slow;
END_REGION

REGION Network 334
   #FP_SIM.WORK.MD_Type_Puls := #FP_SEL.MD_Puls;
END_REGION

REGION Network 335: Adaptor Signals
   #AdapterBlock.Sim_Enable := #TOKEN.Sim_Enable;
END_REGION

REGION Network 336: Flash fast for lamp inidcation
   #AdapterBlock.Flash_Fast := #TOKEN.Flash_Fast;
END_REGION

REGION Network 337: Flash slow for lamp inidcation
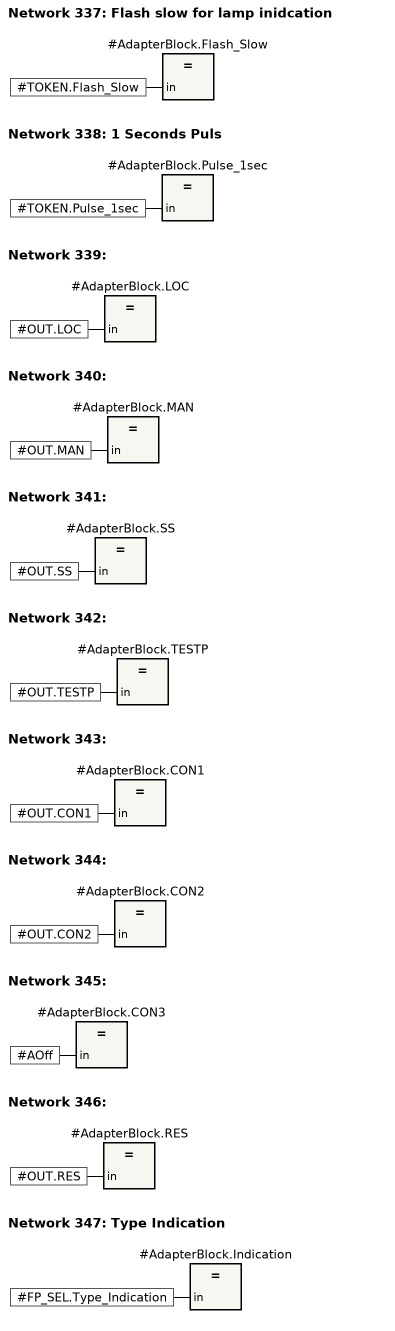
   #AdapterBlock.Flash_Slow := #TOKEN.Flash_Slow;
END_REGION

REGION Network 338: 1 Seconds Puls
   #AdapterBlock.Pulse_1sec := #TOKEN.Pulse_1sec;
END_REGION

REGION Network 339
   #AdapterBlock.LOC := #OUT.LOC;
END_REGION

REGION Network 340
   #AdapterBlock.MAN := #OUT.MAN;
END_REGION

REGION Network 341
   #AdapterBlock.SS := #OUT.SS;
END_REGION

REGION Network 342
   #AdapterBlock.TESTP := #OUT.TESTP;
END_REGION

REGION Network 343
   #AdapterBlock.CON1 := #OUT.CON1;
END_REGION

REGION Network 344
   #AdapterBlock.CON2 := #OUT.CON2;
END_REGION

REGION Network 345
   #AdapterBlock.CON3 := #AOff;
END_REGION

REGION Network 346
   #AdapterBlock.RES := #OUT.RES;
END_REGION

REGION Network 347: Type Indication
   #AdapterBlock.Indication := #FP_SEL.Type_Indication;
END_REGION

REGION Network 348: Write STAT to OUT
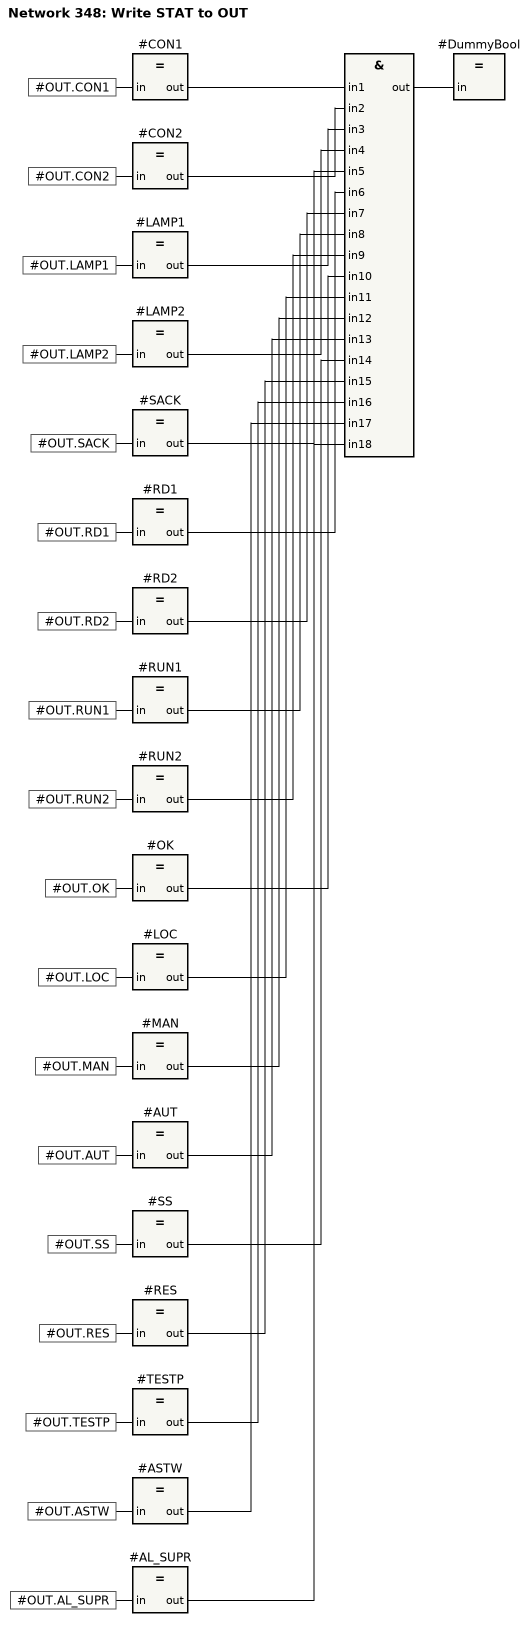
   #CON1 := #OUT.CON1;
   #CON2 := #OUT.CON2;
   #LAMP1 := #OUT.LAMP1;
   #LAMP2 := #OUT.LAMP2;
   #SACK := #OUT.SACK;
   #RD1 := #OUT.RD1;
   #RD2 := #OUT.RD2;
   #RUN1 := #OUT.RUN1;
   #RUN2 := #OUT.RUN2;
   #OK := #OUT.OK;
   #LOC := #OUT.LOC;
   #MAN := #OUT.MAN;
   #AUT := #OUT.AUT;
   #SS := #OUT.SS;
   #RES := #OUT.RES;
   #TESTP := #OUT.TESTP;
   #ASTW := #OUT.ASTW;
   #AL_SUPR := #OUT.AL_SUPR;
   #DummyBool := #OUT.CON1 AND #OUT.CON2 AND #OUT.LAMP1 AND #OUT.LAMP2 AND #OUT.SACK AND #OUT.RD1 AND #OUT.RD2 AND #OUT.RUN1 AND #OUT.RUN2 AND #OUT.OK AND #OUT.LOC AND #OUT.MAN AND #OUT.AUT AND #OUT.SS AND #OUT.RES AND #OUT.TESTP AND #OUT.ASTW AND #OUT.AL_SUPR;
END_REGION
END_FUNCTION_BLOCK

FUNCTION_BLOCK "ACESYS_GATE"   // FB211, FBD
TITLE = ACESYS V8.0 - Build 009 - GATE Block
{ S7_Optimized_Access := 'FALSE' }
AUTHOR : FLSmidth
FAMILY : ACESYS
NAME : GATE
VERSION : 8.0
   VAR_INPUT
      CMD : "ACESYS_GRP_CMD";
      SEL : Bool := TRUE;   // Unit Select by User program
      PREQ1 : Bool := TRUE;   // Direction 1 Select
      PREQ2 : Bool := TRUE;   // Direction 2 Select
      MCC : Bool := TRUE;   // MCC Ready
      RDY : Bool := TRUE;   // Unit ready
      OVL : Bool := TRUE;   // Overload / trip
      RET1 : Bool;   // Feedback contactor 1
      RET2 : Bool;   // Feedback contactor 2
      LSP1 : Bool;   // Limit Switch Pos 1
      LSP2 : Bool;   // Limit Switch Pos 2
      LSA1 : Bool;   // Alarm Switch Pos. 1
      LSA2 : Bool;   // Alarm Switch Pos. 2
      TRQ1 : Bool;   // Torque Switch Pos. 1
      TRQ2 : Bool;   // Torque Switch Pos. 2
      LSTR1 : Bool;   // Local start 1
      LSTR2 : Bool;   // Local start 2
      LSTP : Bool := TRUE;   // Local stop
      REM : Bool := TRUE;   // Unit in Remote operation
      SSW : Bool := TRUE;   // Safety switch
      TFA : Bool := TRUE;   // Termistor fault
      DRDY : Bool := TRUE;   // Drive / MCC ready
      STALL : Bool := TRUE;   // Motor stalled
      EARTH : Bool := TRUE;   // Earth fault
      UBAL : Bool := TRUE;   // Unbalance / Phase lost
      GFA : Bool := TRUE;   // General fault
      GWA : Bool := TRUE;   // General waring
      BUSF : Bool := TRUE;   // Bus failure
      DOPR : Bool := TRUE;   // Drawer in operation position
      DTEST : Bool;   // Drawer in test position
      ACK : Bool;   // Feedback from unit on alarm reset
      POS_OK : Bool;   // Position Signal Healthy
      POS : Real;   // Position Signal
      SP : Real;   // Setpoint
      AI1 : Real;   // Analog value 1
      AI2 : Real;   // Analog value 2
      AI3 : Real;   // Abalog value 3
   END_VAR
   VAR_OUTPUT
      INTL : "ACESYS_INTL";   // Interlock
      INTL_SEQ_STR1 : "ACESYS_INTL";   // Interlock Sequence Start
      INTL_SEQ_STR2 : "ACESYS_INTL";   // Interlock Sequence Start
      INTL_SEQ_STP : "ACESYS_INTL";   // Interlock Sequence Stop
      CON1 : Bool;   // Command 1
      CON2 : Bool;   // Command 2
      LAMP1 : Bool;   // Lamp 1
      LAMP2 : Bool;   // Lamp 2
      SACK : Bool;   // Start Acknowledge
      POS1 : Bool;   // Position 1
      POS2 : Bool;   // Position 2
      RUN1 : Bool;   // Run 1
      RUN2 : Bool;   // Run 2
      OK : Bool;   // Unit Status OK (no alarms)
      LOC : Bool;   // Unit in Local Mode
      MAN : Bool;   // Unit in Manual Mode
      AUT : Bool;   // Unit in Auto Mode
      SS : Bool;   // Unit in Single Start Mode
      RES : Bool;   // Reset to unit
      TESTP : Bool;   // Test mode permission to unit
      ASTW : Bool;   // Start warning
      AL_SUPR : Bool;   // Supress Child Alarms
      AO1a : Real;   // Analog converted 1a
      AO1b : Real;   // Analog converted 1b
      AO2a : Real;   // Analog converted 2a
      AO2b : Real;   // Analog converted 2b
      AO3a : Real;   // Analog converted 3a
      AO3b : Real;   // Analog converted 3b
      MSW : "ACESYS_HMI_STAT_32T";
   END_VAR
   VAR_IN_OUT
      TOKEN : "ACESYS_TOKEN";
   END_VAR
   VAR
      BlockInfo : Struct
         Ace_Version : Int;   // Acesys Block Version Number
         Ace_BuildNo : Int;   // Acesys Block Build Number
         State_Act : Int;   // Actual State Number
         State_Prev : Int;   // Previous State Number
         DB_Number : Int;   // Block Instance DB Number
      END_STRUCT;
      FP_CMD : Struct   // Faceplate Commands
         QuickStop : Bool;
         Spare_09 : Bool;
         Spare_10 : Bool;
         Spare_11 : Bool;
         Spare_12 : Bool;
         Spare_13 : Bool;
         Spare_14 : Bool;
         AckAlarm : Bool;
         Auto : Bool;
         Manual : Bool;
         Local : Bool;
         Start1 : Bool;
         Start2 : Bool;
         Stop : Bool;
         Reset : Bool;
         Test : Bool;
      END_STRUCT;
      FP_SEL : Struct   // Faceplate Selections
         STW_AutoStart : Bool;   // Faceplate Start Warning in Auto Start mode
         STW_Local : Bool;   // Faceplate Start Warning in Local mode
         STW_Manual : Bool;   // Faceplate Start Warning in Manual mode
         STW_Single : Bool;   // Faceplate Start Warning in Single Start mode
         Type_MotorGate : Bool;   // Faceplate Motorgate type
         Type_Positioner : Bool;   // Faceplate Positioner type
         Type_Indication : Bool;   // Faceplate Indication type
         ParentSupress : Bool;   // Enable Parent Supress of alarms
         ParentCollection : Bool;   // Enable Inching in Manual Mode
         INCH_Man : Bool;   // Enable Inching in Manual Mode
         INCH_Loc : Bool;   // Enable Inching in Local Mode
         OutOfSevice : Bool;   // Select Out of Service
         WarningDrive : Bool;   // 0 = Failure Drive / 1 = Warning Drive
         Park_CurrPos : Bool;
         Park_Pos1 : Bool;
         Park_Pos2 : Bool;
         GroupMode : Bool;
         GroupCtrl : Bool;
         Spare14 : Bool;
         Spare13 : Bool;
         Spare12 : Bool;
         Spare11 : Bool;
         Spare10 : Bool;
         Spare9 : Bool;
         Spare8 : Bool;
         Spare7 : Bool;
         Spare6 : Bool;
         Spare5 : Bool;
         Spare4 : Bool;
         Spare3 : Bool;
         Spare2 : Bool;
         Spare1 : Bool;
      END_STRUCT;
      FP_EN : Struct
         Mode_Auto : Bool;
         Mode_Man : Bool;
         Mode_Loc : Bool;
         Mode_Test : Bool;
         Mode_SS_Field : Bool;
         Mode_SS_FP : Bool;
         PB_QStop : Bool;
         Wagging : Bool;   // Wagging
         Spare8 : Bool;
         Spare7 : Bool;
         Spare6 : Bool;
         Spare5 : Bool;
         Spare4 : Bool;
         Spare3 : Bool;
         Spare2 : Bool;
         Spare1 : Bool;
      END_STRUCT;
      FP_DIM : Struct   // Faceplate Dimmed Buttons
         Auto : Bool;
         Local : Bool;
         Manual : Bool;
         Start1 : Bool;
         Start2 : Bool;
         Stop : Bool;
         Test : Bool;
         QStop : Bool;
         Reset : Bool;
         Spare7 : Bool;
         Spare6 : Bool;
         Spare5 : Bool;
         Spare4 : Bool;
         Spare3 : Bool;
         Spare2 : Bool;
         Spare1 : Bool;
      END_STRUCT;
      FP_SHOW : Struct   // Faceplate Show Buttons
         PB_Auto : Bool;
         PB_Local : Bool;
         PB_Manual : Bool;
         PB_Start1 : Bool;
         PB_Start2 : Bool;
         PB_Stop : Bool;
         PB_Test : Bool;
         PB_QStop : Bool;
         AI1 : Bool;
         AI2 : Bool;
         AI3 : Bool;
         MCC : Bool;
         RDY : Bool;
         OVL : Bool;
         LSTP : Bool;
         REM : Bool;
         SSW : Bool;
         Spare : Bool;
         TFA : Bool;
         DRDY : Bool;
         STALL : Bool;
         EARTH : Bool;
         UBAL : Bool;
         GFA : Bool;
         GWA : Bool;
         BUSF : Bool;
         DOPR : Bool;
         DTEST : Bool;
         ACK : Bool;
         LSTR1 : Bool;
         LSTR2 : Bool;
         LSA1 : Bool;
         LSA2 : Bool;
         TRQ1 : Bool;
         TRQ2 : Bool;
         PB_Reset : Bool;
         Spare4 : Bool;
         Spare3 : Bool;
         Spare2 : Bool;
         Spare1 : Bool;
      END_STRUCT;
      FP_PARM : Struct   // Faceplate Parameters
         StartWarn_Pre : Int;
         StartWarn_Acc : Int;
         RunTime_Pre : Int;
         RunTime_Acc : Int;
         DriftingTime_Pre : Int;
         DriftingTime_Acc : Int;
         DelayStart_Pre : Int;
         DelayStart_Acc : Int;
         DelayStop_Pre : Int;
         DelayStop_Acc : Int;
         ReturnMon_Pre : Int;
         ReturnMon_Acc : Int;
         ChangeDir_Pre : Int;
         ChangeDir_Acc : Int;
         WaitTime_Pre : Int;
         WaitTime_Acc : Int;
         Wagging_Pre : Int;
         Wagging_Acc : Int;
         RunTimeActuator : Real := 60.0;
         DeadBand : Real := 1.5;
         Sensibility : Real := 97.0;
         MinPulsetime : Int;
         AI1_Max : Real;
         AI1_Min : Real;
         AI2_Max : Real;
         AI2_Min : Real;
         AI3_Max : Real;
         AI3_Min : Real;
         AO1a_Max : Real;
         AO1a_Min : Real;
         AO2a_Max : Real;
         AO2a_Min : Real;
         AO3a_Max : Real;
         AO3a_Min : Real;
         AO1b_Max : Real;
         AO1b_Min : Real;
         AO2b_Max : Real;
         AO2b_Min : Real;
         AO3b_Max : Real;
         AO3b_Min : Real;
         INTL : Bool;   // Interlock
         INTL_SEQ_STR1 : Bool;   // Interlock Sequence Start
         INTL_SEQ_STR2 : Bool;   // Interlock Sequence Start
         INTL_SEQ_STP : Bool;   // Interlock Sequence Stop
         Spare12 : Bool;
         Spare11 : Bool;
         Spare10 : Bool;
         Spare09 : Bool;
         Spare08 : Bool;
         Spare07 : Bool;
         Spare06 : Bool;
         Spare05 : Bool;
         Spare04 : Bool;
         Spare03 : Bool;
         Spare02 : Bool;
         Spare01 : Bool;
      END_STRUCT;
      FP_SIM : "ACESYS_SIM_GATE";
      AdapterBlock : "ACESYS_ADPT_MOTOR";
      STATE : Struct
         A_Ctrl_AutoStart : Bool;
         A_Ctrl_DelayedStart1 : Bool;
         A_Ctrl_DelayedStart2 : Bool;
         A_Ctrl_DelayedStop : Bool;
         A_Ctrl_MoveToPos1 : Bool;
         A_Ctrl_MoveToPos2 : Bool;
         A_Ctrl_Parking1 : Bool;
         A_Ctrl_Parking2 : Bool;
         A_Ctrl_ParkStartWarning : Bool;
         A_Ctrl_Pos1 : Bool;
         A_Ctrl_Pos2 : Bool;
         A_Ctrl_Selected : Bool;
         A_Ctrl_SelToStop : Bool;
         A_Ctrl_SeqStart1 : Bool;
         A_Ctrl_SeqStart2 : Bool;
         A_Ctrl_SeqStop : Bool;
         A_Ctrl_Starting1 : Bool;
         A_Ctrl_Starting2 : Bool;
         A_Ctrl_StartWarning1 : Bool;
         A_Ctrl_StartWarning2 : Bool;
         A_Ctrl_Stopped : Bool;
         A_Ctrl_Stopping : Bool;
         A_Ctrl_WaggingToPos1 : Bool;
         A_Ctrl_WaggingToPos2 : Bool;
         A_NoCtrl_AutoStart : Bool;
         A_NoCtrl_Pos1 : Bool;
         A_NoCtrl_Pos2 : Bool;
         A_NoCtrl_MoveToPos1 : Bool;
         A_NoCtrl_MoveToPos2 : Bool;
         A_NoCtrl_SeqStart1 : Bool;
         A_NoCtrl_SeqStart2 : Bool;
         A_NoCtrl_Starting1 : Bool;
         A_NoCtrl_Starting2 : Bool;
         A_NoCtrl_StartWarning1 : Bool;
         A_NoCtrl_StartWarning2 : Bool;
         A_NoCtrl_WaggingToPos1 : Bool;
         A_NoCtrl_WaggingToPos2 : Bool;
         S_AutoStart : Bool;
         S_MoveToPos1 : Bool;
         S_MoveToPos2 : Bool;
         S_NotActive : Bool;
         S_Parking1 : Bool;
         S_Parking2 : Bool;
         S_ParkStartWarning : Bool;
         S_Pos1 : Bool;
         S_Pos2 : Bool;
         S_Starting1 : Bool;
         S_Starting2 : Bool;
         S_StartWarning1 : Bool;
         S_StartWarning2 : Bool;
         S_Stopping : Bool;
         S_WaggingToPos1 : Bool;
         S_WaggingToPos2 : Bool;
         M_AutoStart : Bool;
         M_MoveToPos1 : Bool;
         M_MoveToPos2 : Bool;
         M_NotActive : Bool;
         M_Pos1 : Bool;
         M_Pos2 : Bool;
         M_Starting1 : Bool;
         M_Starting2 : Bool;
         M_StartWarning1 : Bool;
         M_StartWarning2 : Bool;
         L_AutoStart : Bool;
         L_MoveToPos1 : Bool;
         L_MoveToPos2 : Bool;
         L_NotActive : Bool;
         L_Pos1 : Bool;
         L_Pos2 : Bool;
         L_Starting1 : Bool;
         L_Starting2 : Bool;
         L_StartWarning1 : Bool;
         L_StartWarning2 : Bool;
         T_Starting1 : Bool;
         T_Starting2 : Bool;
         T_TestMode : Bool;
         T_TestPermission : Bool;
         Alarm : Bool;
         Interlock : Bool;
         EmergencyStop : Bool;
         OutOfService : Bool;
      END_STRUCT;
      ONS : Struct
         Motorgate : Bool;
         Positioner : Bool;
         LSTR1_1 : Bool;
         LSTR1_2 : Bool;
         LSTR2_1 : Bool;
         LSTR2_2 : Bool;
         AckAlarm : Bool;
         Cmd_Auto : Bool;
         Cmd_Manual : Bool;
         CMD_Local : Bool;
         CMD_Test : Bool;
         GLTP : Bool;
         MasterStop : Bool;
         RET1 : Bool;
         RET2 : Bool;
         Park_Curr : Bool;
         Park_Pos1 : Bool;
         Park_Pos2 : Bool;
         Wagging : Bool;
         Recalc : Bool;
         FP_Start1_CMD : Bool;
         FP_Start2_CMD : Bool;
         CMD_Start1 : Bool;
         CMD_Start2 : Bool;
         SecPulse1 : Bool;
         SecPulse2 : Bool;
         GSS_On : Bool;
         Spare5 : Bool;
         Spare4 : Bool;
         Spare3 : Bool;
         Spare2 : Bool;
         Spare1 : Bool;
      END_STRUCT;
      StatusWork : Int;
      ModePointer : Int;
      AlarmNo : Int;
      AlarmNo_Old : Int;
      StartWarn_Mem : Int;
      Runtime_Mem : Int;
      DriftingTime_Mem : Int;
      WaitTime_Mem : Int;
      DelayStart_Mem : Int;
      DelayStop_Mem : Int;
      ReturnMon_Mem : Int;
      ChangeDir1_Mem : Int;
      ChangeDir2_Mem : Int;
      CalcPosRuntime_DINT : DInt;
      Difference_ABS : Real;
      Old_SP : Real;
      ModeAuto : Bool;
      ModeLocal : Bool;
      ModeManual : Bool;
      ModeSingleStart : Bool;
      ModeTest : Bool;
      Select : Bool;   // Parent & Program Select
      CMD_AckAlarm : Bool;
      CMD_Start1 : Bool;
      CMD_Start2 : Bool;
      CMD_Stop : Bool;
      CMD_QStop : Bool;
      CMD_Reset : Bool;
      FromStateAuto : Bool;
      FromStateAuto_GrpCtrl : Bool;
      FromStateAuto_NoGrpCtrl : Bool;
      FromStateSingle : Bool;
      FromStateManual : Bool;
      FromStateLocal : Bool;
      FromStateTest : Bool;
      FromStopState : Bool;
      ALARM_SupressionActive : Bool;
      ALARM_AlarmPresent : Bool;
      ALARM_WarnPresent : Bool;
      ALARM_FailureAckRequired : Bool;
      ALARM_WarnAckRequired : Bool;
      StartWarn_TT : Bool;
      StartWarn_Done : Bool;
      WaitTime_TT : Bool;
      WaitTime_Done : Bool;
      RunTime_Done : Bool;
      DriftingTime_Done : Bool;
      DelayStart_Done : Bool;
      DelayStop_Done : Bool;
      ReturnMon_Done : Bool;
      ChangeDir1_Done : Bool;
      ChangeDir2_Done : Bool;
      ChangeDir1_TT : Bool;
      ChangeDir2_TT : Bool;
      Timer_Position_Done : Bool;
      Trig_ALARM_RET : Bool;
      Trig_ALARM_Runtime : Bool;
      Trig_ALARM_Drifting : Bool;
      RET1_OneScan : Bool;
      RET2_OneScan : Bool;
      LSTR1_Puls : Bool;
      LSTR2_Puls : Bool;
      DIR1_Request : Bool;
      DIR2_Request : Bool;
      Request_Up : Bool;
      Request_Down : Bool;
      Recalculate : Bool;
      LimitDrifting1 : Bool;
      LimitDrifting2 : Bool;
      LimitSwitchPos1Mem : Bool;
      LimitSwitchPos2Mem : Bool;
      CountElapsed_Wagging : Bool;
      OK_Alarm : Bool;
      SpareBool_7 : Bool;
      SpareBool_6 : Bool;
      SpareBool_5 : Bool;
      SpareBool_4 : Bool;
      SpareBool_3 : Bool;
      SpareBool_2 : Bool;
      SpareBool_1 : Bool;
      Sec_Pulse : Bool;
      Timer_Position : TON_TIME;
      Timer_Positioner_PRE : Time;
      OUT : Struct
         CON1 : Bool;
         CON2 : Bool;
         LAMP1 : Bool;
         LAMP2 : Bool;
         SACK : Bool;
         POS1 : Bool;
         POS2 : Bool;
         RUN1 : Bool;
         RUN2 : Bool;
         OK : Bool;
         LOC : Bool;
         MAN : Bool;
         AUT : Bool;
         SS : Bool;
         RES : Bool;
         TESTP : Bool;
         ASTW : Bool;
         AL_SUPR : Bool;
         INTL_OK_STAT : Bool;
         INTL_SEQ_STR1_OK_STAT : Bool;
         INTL_SEQ_STR2_OK_STAT : Bool;
         INTL_SEQ_STP_OK_STAT : Bool;
         MSW_EXT_ALARMFAILUNACK : Bool;
      END_STRUCT;
      MSW_Status_Trans : Int;
   END_VAR
   VAR_TEMP
      AOn : Bool;   // Always On
      AOff : Bool;   // Always Off
      DummyBool : Bool;
      StatPointer_Old : Int;
      ChangeDir1_Acc : Int;
      ChangeDir2_Acc : Int;
      StatusBuilder : Int;
      helpReal : Real;
      Timer_Positioner_ACC : Time;
      Difference : Real;
      MinPulsLengt_DINT : DInt;
      Status_Add : Int;
   END_VAR
   VAR_TEMP   // added for the SCL form of the ladder/FBD networks
      _w1 : Bool;
      _w2 : Bool;
      _w3 : Bool;
      _w4 : Bool;
      _w5 : Bool;
      _w6 : Bool;
      _w7 : Bool;
      _w8 : Bool;
   END_VAR
BEGIN

REGION Network 1: Always On
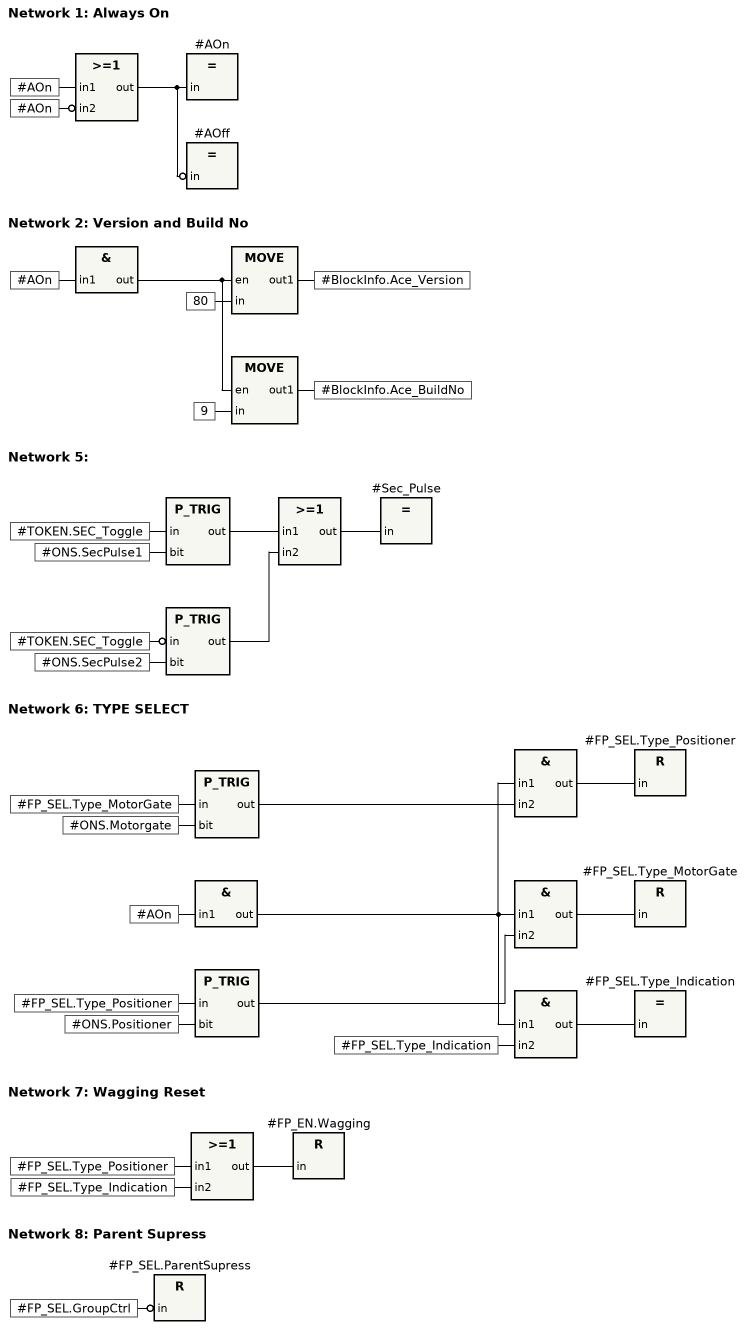
   #AOn := #AOn OR NOT #AOn;
   #AOff := NOT #AOn;
END_REGION

REGION Network 2: Version and Build No
   IF #AOn THEN
       #BlockInfo.Ace_Version := 80;
       #BlockInfo.Ace_BuildNo := 9;
   END_IF;
END_REGION

REGION Network 3 (STL): Instance DB Number to Faceplate
         L     DINO;
         T     #BlockInfo.DB_Number;
END_REGION

REGION Network 4 (SCL): Transfer Interlock OK to Stat
   #OUT.INTL_OK_STAT := PEEK_BOOL(area := 16#84, dbNumber := #BlockInfo.DB_Number, byteOffset := 26, bitOffset := 0);
   #OUT.INTL_SEQ_STR1_OK_STAT := PEEK_BOOL(area := 16#84, dbNumber := #BlockInfo.DB_Number, byteOffset := 28, bitOffset := 0);
   #OUT.INTL_SEQ_STR2_OK_STAT := PEEK_BOOL(area := 16#84, dbNumber := #BlockInfo.DB_Number, byteOffset := 30, bitOffset := 0);
   #OUT.INTL_SEQ_STP_OK_STAT := PEEK_BOOL(area := 16#84, dbNumber := #BlockInfo.DB_Number, byteOffset := 32, bitOffset := 0);
END_REGION

REGION Network 5
   #_w1 := #TOKEN.SEC_Toggle AND NOT #ONS.SecPulse1;   // rising edge
   #ONS.SecPulse1 := #TOKEN.SEC_Toggle;
   #_w2 := NOT #TOKEN.SEC_Toggle AND NOT #ONS.SecPulse2;   // rising edge
   #ONS.SecPulse2 := NOT #TOKEN.SEC_Toggle;
   #Sec_Pulse := #_w1 OR #_w2;
END_REGION

REGION Network 6: TYPE SELECT
   #_w1 := #FP_SEL.Type_MotorGate AND NOT #ONS.Motorgate;   // rising edge
   #ONS.Motorgate := #FP_SEL.Type_MotorGate;
   IF #AOn AND #_w1 THEN #FP_SEL.Type_Positioner := FALSE; END_IF;
   #_w2 := #FP_SEL.Type_Positioner AND NOT #ONS.Positioner;   // rising edge
   #ONS.Positioner := #FP_SEL.Type_Positioner;
   IF #AOn AND #_w2 THEN #FP_SEL.Type_MotorGate := FALSE; END_IF;
   #FP_SEL.Type_Indication := #AOn AND #FP_SEL.Type_Indication;
END_REGION

REGION Network 7: Wagging Reset
   IF #FP_SEL.Type_Positioner OR #FP_SEL.Type_Indication THEN #FP_EN.Wagging := FALSE; END_IF;
END_REGION

REGION Network 8: Parent Supress
   IF NOT #FP_SEL.GroupCtrl THEN #FP_SEL.ParentSupress := FALSE; END_IF;
END_REGION

REGION Network 9: Status Update
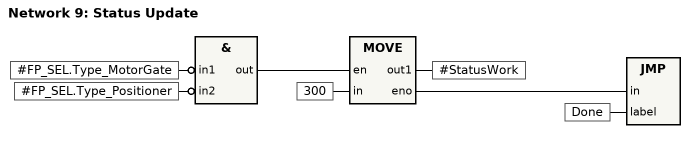
   // ENO of a box is taken as its EN; it also drops when the box reports an error
   #_w1 := NOT #FP_SEL.Type_MotorGate AND NOT #FP_SEL.Type_Positioner;
   IF #_w1 THEN
       #StatusWork := 300;
       GOTO Done;
   END_IF;
END_REGION

REGION Network 10: SET SHOW PARAMETERS
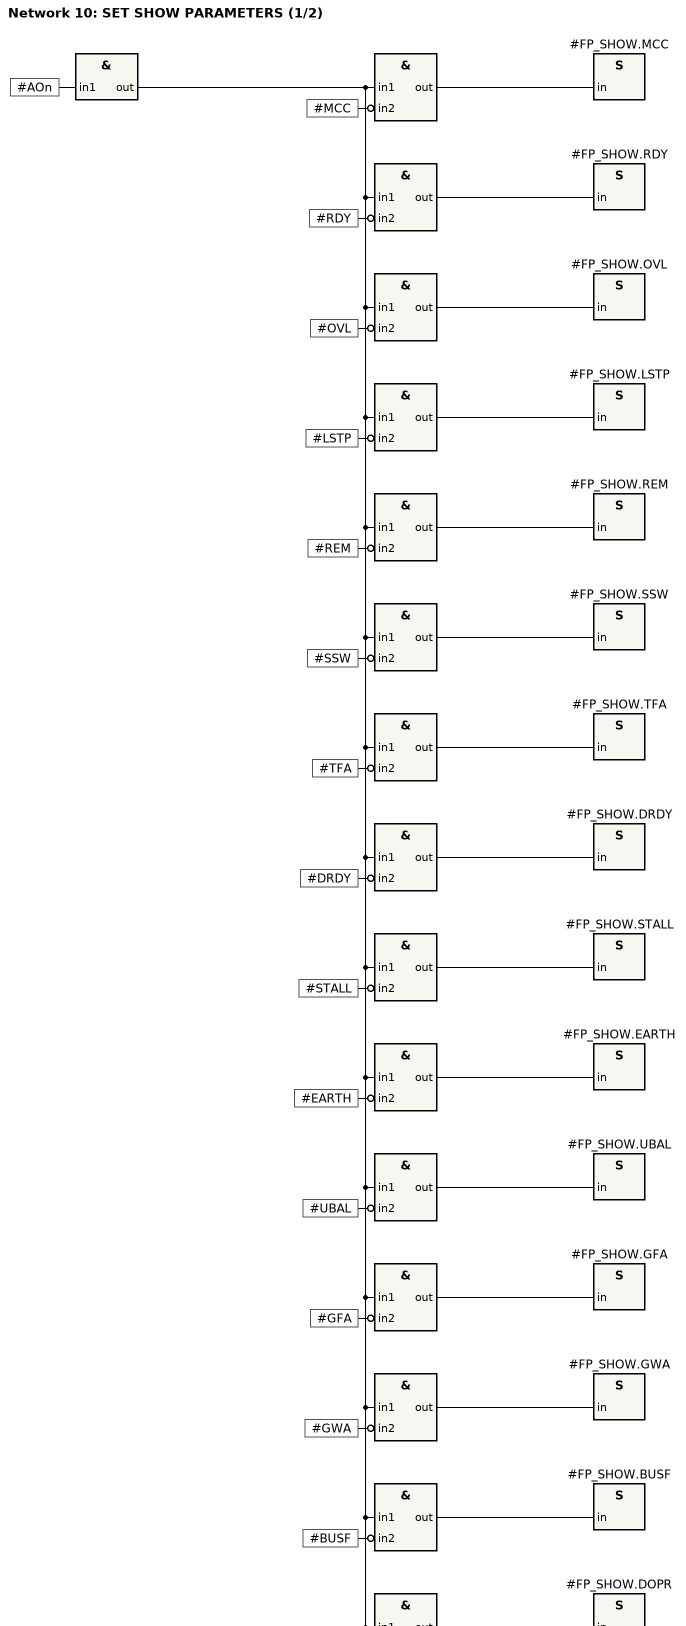
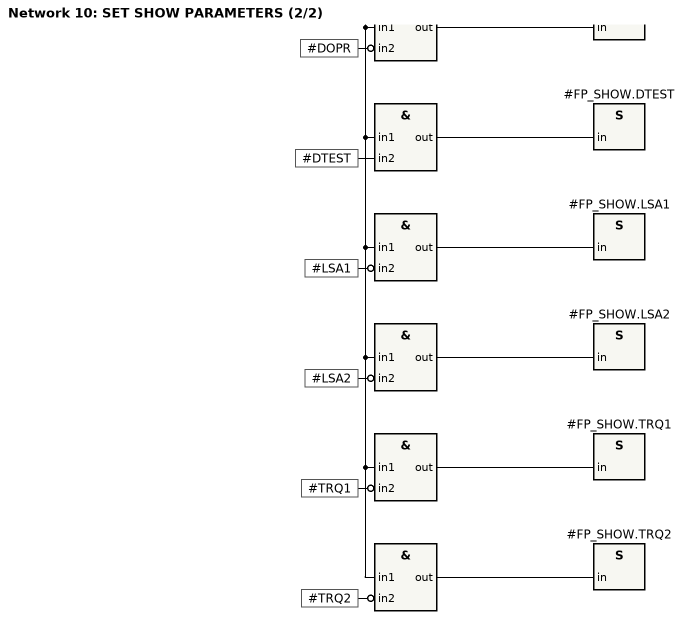
   IF #AOn AND NOT #MCC THEN #FP_SHOW.MCC := TRUE; END_IF;
   IF #AOn AND NOT #RDY THEN #FP_SHOW.RDY := TRUE; END_IF;
   IF #AOn AND NOT #OVL THEN #FP_SHOW.OVL := TRUE; END_IF;
   IF #AOn AND NOT #LSTP THEN #FP_SHOW.LSTP := TRUE; END_IF;
   IF #AOn AND NOT #REM THEN #FP_SHOW.REM := TRUE; END_IF;
   IF #AOn AND NOT #SSW THEN #FP_SHOW.SSW := TRUE; END_IF;
   IF #AOn AND NOT #TFA THEN #FP_SHOW.TFA := TRUE; END_IF;
   IF #AOn AND NOT #DRDY THEN #FP_SHOW.DRDY := TRUE; END_IF;
   IF #AOn AND NOT #STALL THEN #FP_SHOW.STALL := TRUE; END_IF;
   IF #AOn AND NOT #EARTH THEN #FP_SHOW.EARTH := TRUE; END_IF;
   IF #AOn AND NOT #UBAL THEN #FP_SHOW.UBAL := TRUE; END_IF;
   IF #AOn AND NOT #GFA THEN #FP_SHOW.GFA := TRUE; END_IF;
   IF #AOn AND NOT #GWA THEN #FP_SHOW.GWA := TRUE; END_IF;
   IF #AOn AND NOT #BUSF THEN #FP_SHOW.BUSF := TRUE; END_IF;
   IF #AOn AND NOT #DOPR THEN #FP_SHOW.DOPR := TRUE; END_IF;
   IF #AOn AND #DTEST THEN #FP_SHOW.DTEST := TRUE; END_IF;
   IF #AOn AND NOT #LSA1 THEN #FP_SHOW.LSA1 := TRUE; END_IF;
   IF #AOn AND NOT #LSA2 THEN #FP_SHOW.LSA2 := TRUE; END_IF;
   IF #AOn AND NOT #TRQ1 THEN #FP_SHOW.TRQ1 := TRUE; END_IF;
   IF #AOn AND NOT #TRQ2 THEN #FP_SHOW.TRQ2 := TRUE; END_IF;
END_REGION

REGION Network 11: SET SHOW PARAMETERS
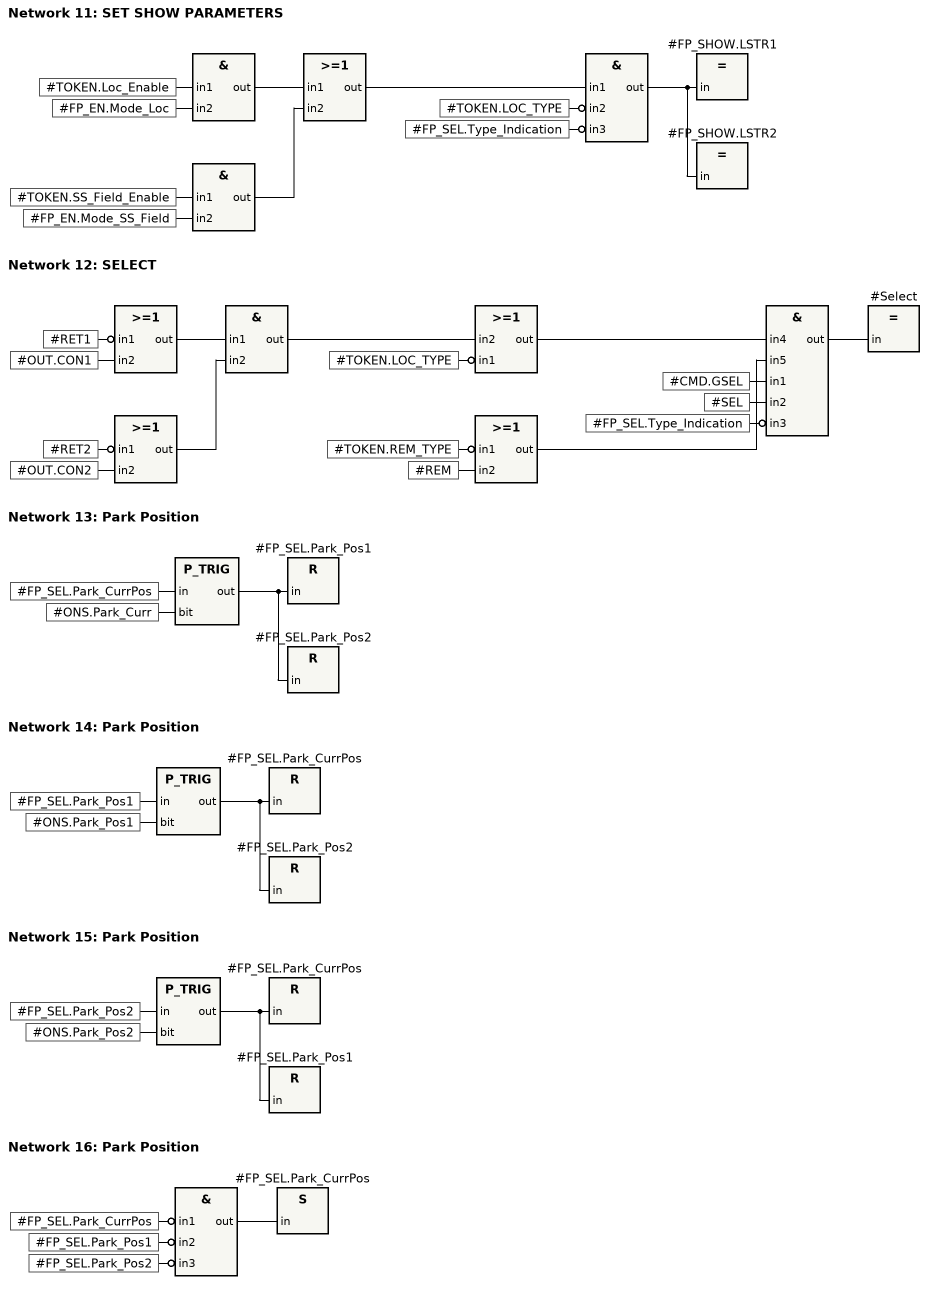
   #FP_SHOW.LSTR1 := ((#TOKEN.Loc_Enable AND #FP_EN.Mode_Loc) OR (#TOKEN.SS_Field_Enable AND #FP_EN.Mode_SS_Field)) AND NOT #TOKEN.LOC_TYPE AND NOT #FP_SEL.Type_Indication;
   #FP_SHOW.LSTR2 := #FP_SHOW.LSTR1;
END_REGION

REGION Network 12: SELECT
   // Build 003 - 2.July.2019 (EXTBOB): Added logic to prevent group selection interference when gate is running in "electrical" local mode or mode is controlled from the field.
   #Select := (((NOT #RET1 OR #OUT.CON1) AND (NOT #RET2 OR #OUT.CON2)) OR NOT #TOKEN.LOC_TYPE) AND (NOT #TOKEN.REM_TYPE OR #REM) AND #CMD.GSEL AND #SEL AND NOT #FP_SEL.Type_Indication;
END_REGION

REGION Network 13: Park Position
   #_w1 := #FP_SEL.Park_CurrPos AND NOT #ONS.Park_Curr;   // rising edge
   #ONS.Park_Curr := #FP_SEL.Park_CurrPos;
   IF #_w1 THEN
       #FP_SEL.Park_Pos1 := FALSE;
       #FP_SEL.Park_Pos2 := FALSE;
   END_IF;
END_REGION

REGION Network 14: Park Position
   #_w1 := #FP_SEL.Park_Pos1 AND NOT #ONS.Park_Pos1;   // rising edge
   #ONS.Park_Pos1 := #FP_SEL.Park_Pos1;
   IF #_w1 THEN
       #FP_SEL.Park_CurrPos := FALSE;
       #FP_SEL.Park_Pos2 := FALSE;
   END_IF;
END_REGION

REGION Network 15: Park Position
   #_w1 := #FP_SEL.Park_Pos2 AND NOT #ONS.Park_Pos2;   // rising edge
   #ONS.Park_Pos2 := #FP_SEL.Park_Pos2;
   IF #_w1 THEN
       #FP_SEL.Park_CurrPos := FALSE;
       #FP_SEL.Park_Pos1 := FALSE;
   END_IF;
END_REGION

REGION Network 16: Park Position
   IF NOT #FP_SEL.Park_CurrPos AND NOT #FP_SEL.Park_Pos1 AND NOT #FP_SEL.Park_Pos2 THEN
       #FP_SEL.Park_CurrPos := TRUE;
   END_IF;
END_REGION

REGION Network 17: Group Mode
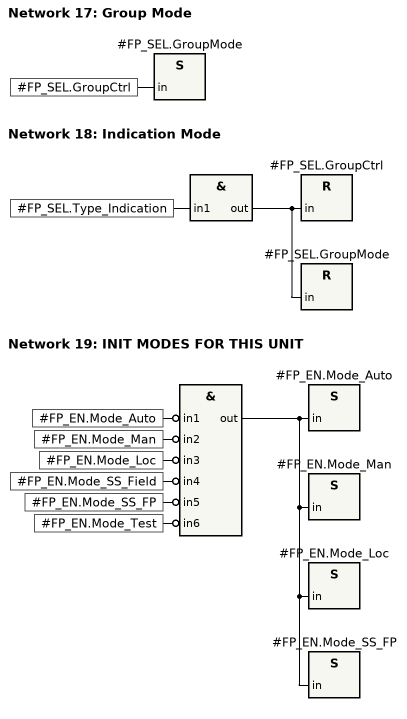
   IF #FP_SEL.GroupCtrl THEN #FP_SEL.GroupMode := TRUE; END_IF;
END_REGION

REGION Network 18: Indication Mode
   IF #FP_SEL.Type_Indication THEN
       #FP_SEL.GroupCtrl := FALSE;
       #FP_SEL.GroupMode := FALSE;
   END_IF;
END_REGION

REGION Network 19: INIT MODES FOR THIS UNIT
   #_w1 := NOT #FP_EN.Mode_Auto AND NOT #FP_EN.Mode_Man AND NOT #FP_EN.Mode_Loc AND NOT #FP_EN.Mode_SS_Field AND NOT #FP_EN.Mode_SS_FP AND NOT #FP_EN.Mode_Test;
   IF #_w1 THEN
       #FP_EN.Mode_Auto := TRUE;
       #FP_EN.Mode_Man := TRUE;
       #FP_EN.Mode_Loc := TRUE;
       #FP_EN.Mode_SS_FP := TRUE;
   END_IF;
END_REGION

REGION Network 20: SHOW PUSH BUTTONS ON FACEPLATE
   // Build 002 - 26 March 2019 : LOC_Type flag removed from Show_PB_local
   // Build 002 - 26 March 2019 : En_Mode_Test flag added in PB_Start1/2 & PB_Stop
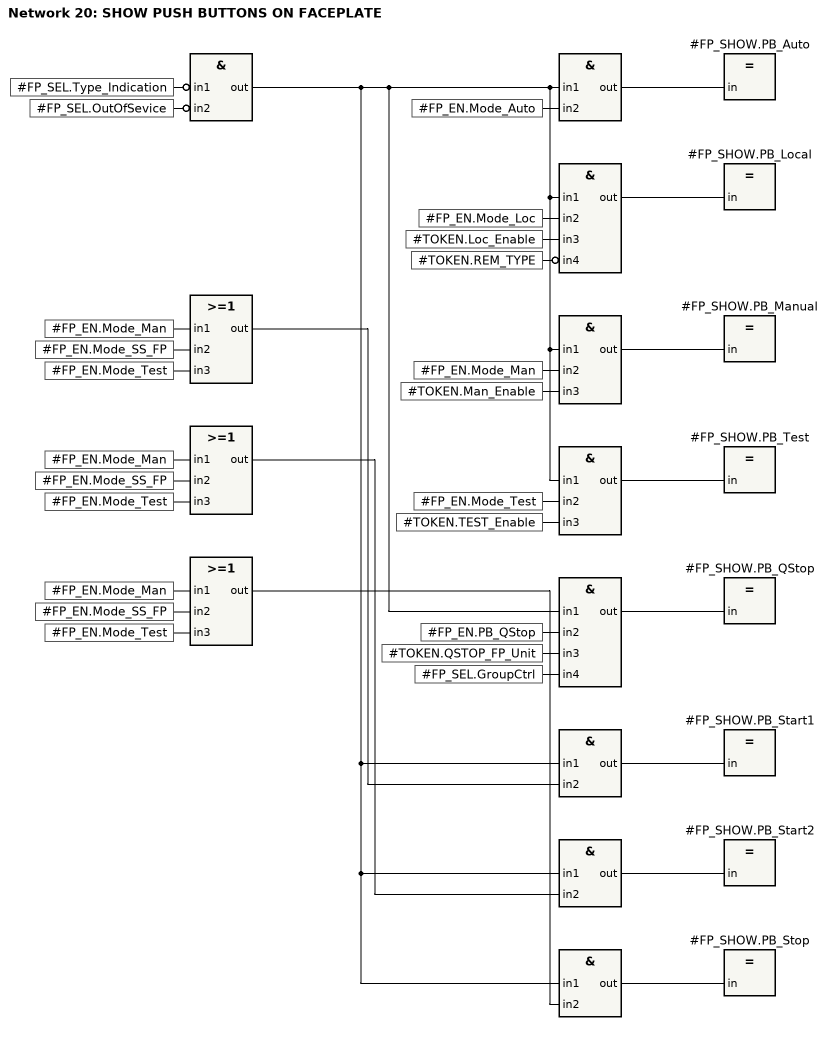
   #_w1 := NOT #FP_SEL.Type_Indication AND NOT #FP_SEL.OutOfSevice;
   #FP_SHOW.PB_Auto := #_w1 AND #FP_EN.Mode_Auto;
   #FP_SHOW.PB_Local := #_w1 AND #FP_EN.Mode_Loc AND #TOKEN.Loc_Enable AND NOT #TOKEN.REM_TYPE;
   #FP_SHOW.PB_Manual := #_w1 AND #FP_EN.Mode_Man AND #TOKEN.Man_Enable;
   #FP_SHOW.PB_Test := #_w1 AND #FP_EN.Mode_Test AND #TOKEN.TEST_Enable;
   #FP_SHOW.PB_QStop := #_w1 AND #FP_EN.PB_QStop AND #TOKEN.QSTOP_FP_Unit AND #FP_SEL.GroupCtrl;
   #FP_SHOW.PB_Start1 := #_w1 AND (#FP_EN.Mode_Man OR #FP_EN.Mode_SS_FP OR #FP_EN.Mode_Test);
   #FP_SHOW.PB_Start2 := #_w1 AND (#FP_EN.Mode_Man OR #FP_EN.Mode_SS_FP OR #FP_EN.Mode_Test);
   #FP_SHOW.PB_Stop := #_w1 AND (#FP_EN.Mode_Man OR #FP_EN.Mode_SS_FP OR #FP_EN.Mode_Test);
END_REGION

REGION Network 21: DIMOUT AUTO BUTTON ON FACEPLATE
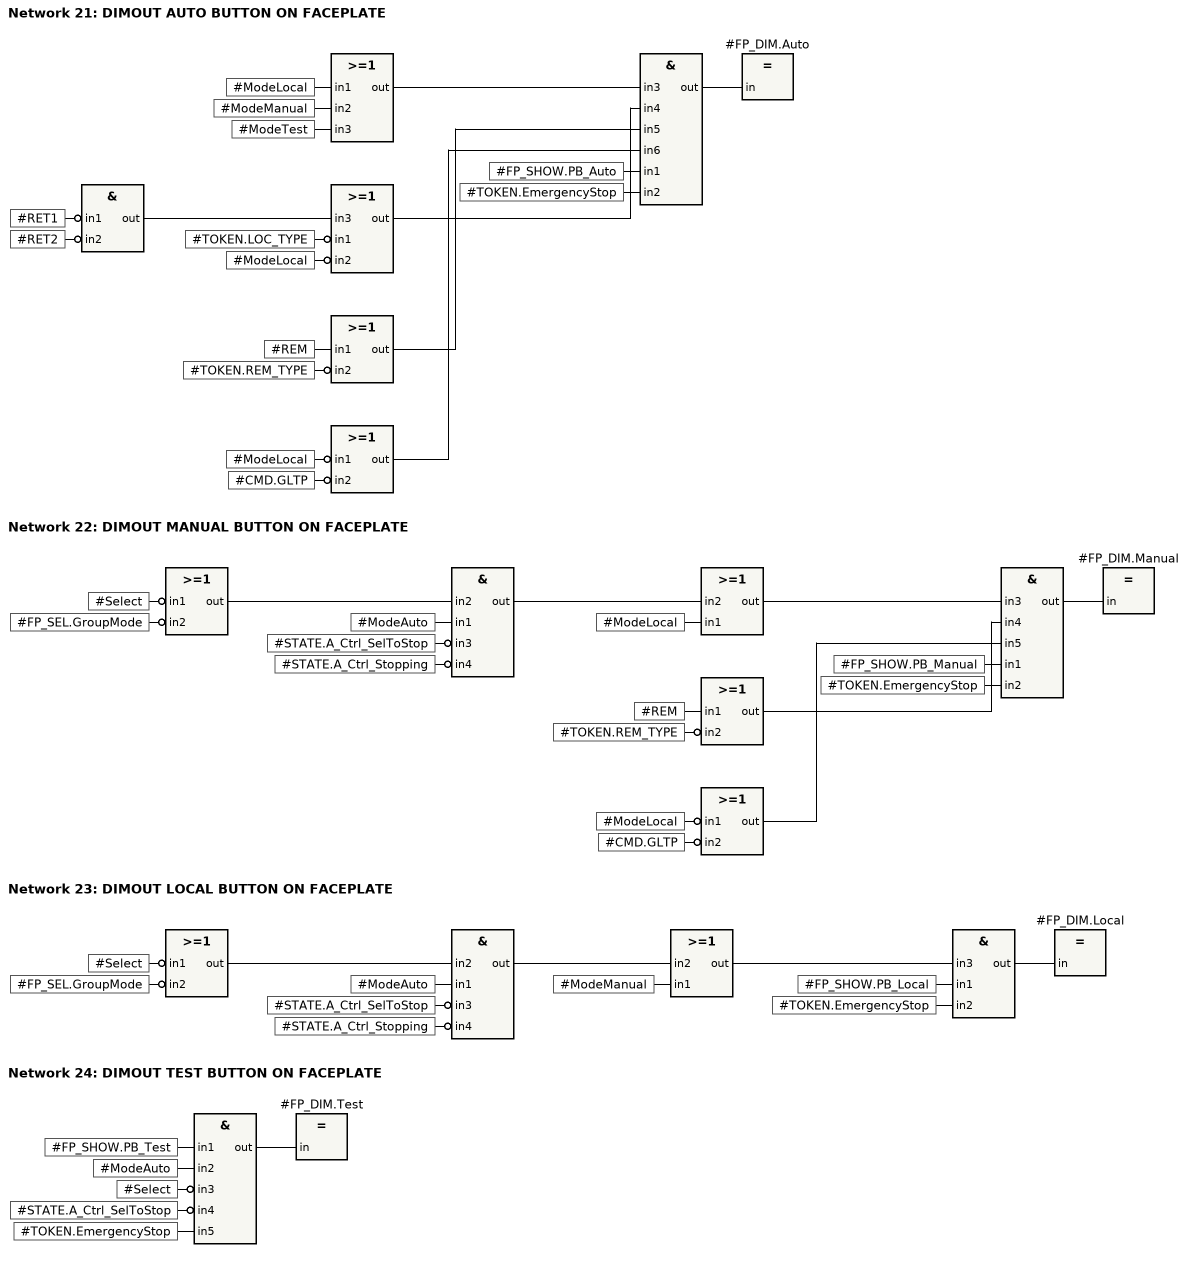
   #FP_DIM.Auto := (#ModeLocal OR #ModeManual OR #ModeTest) AND ((NOT #RET1 AND NOT #RET2) OR NOT #TOKEN.LOC_TYPE OR NOT #ModeLocal) AND (#REM OR NOT #TOKEN.REM_TYPE) AND (NOT #ModeLocal OR NOT #CMD.GLTP) AND #FP_SHOW.PB_Auto AND #TOKEN.EmergencyStop;
END_REGION

REGION Network 22: DIMOUT MANUAL BUTTON ON FACEPLATE
   #FP_DIM.Manual := (((NOT #Select OR NOT #FP_SEL.GroupMode) AND #ModeAuto AND NOT #STATE.A_Ctrl_SelToStop AND NOT #STATE.A_Ctrl_Stopping) OR #ModeLocal) AND (#REM OR NOT #TOKEN.REM_TYPE) AND (NOT #ModeLocal OR NOT #CMD.GLTP) AND #FP_SHOW.PB_Manual AND #TOKEN.EmergencyStop;
END_REGION

REGION Network 23: DIMOUT LOCAL BUTTON ON FACEPLATE
   #FP_DIM.Local := (((NOT #Select OR NOT #FP_SEL.GroupMode) AND #ModeAuto AND NOT #STATE.A_Ctrl_SelToStop AND NOT #STATE.A_Ctrl_Stopping) OR #ModeManual) AND #FP_SHOW.PB_Local AND #TOKEN.EmergencyStop;
END_REGION

REGION Network 24: DIMOUT TEST BUTTON ON FACEPLATE
   #FP_DIM.Test := #FP_SHOW.PB_Test AND #ModeAuto AND NOT #Select AND NOT #STATE.A_Ctrl_SelToStop AND #TOKEN.EmergencyStop;
END_REGION

REGION Network 25: DIMOUT STOP BUTTON ON FACEPLATE
